// TIA Portal project "sorting and packaging f" (V16)
// Vorlageprojekt für das Buch mit Zielsystem S7-1200

(* hardware
DEVICE "S7-1200-Station_1"  S7-1200 Station
   slot 0: "Baugruppenträger_0"  Rack  V1.0
   slot 1: "PLC_1"  CPU 1211C DC/DC/DC  6ES7 211-1AE40-0XB0  V4.1
*)

// ===== PLC "PLC_1"  CPU 1211C DC/DC/DC =====

VAR_GLOBAL   // PLC tag table "Standard-Variablentabelle"
   "start" AT %I0.0 : Bool;
   "stop" AT %I0.1 : Bool;
   "emergency" AT %I0.2 : Bool;
   "vision1" AT %ID30 : DInt;
   "diff1" AT %I0.4 : Bool;
   "zdownsens1" AT %I0.5 : Bool;
   "box1" AT %I0.7 : Bool;
   "xmovesens1" AT %I1.0 : Bool;
   "rotate1" AT %I1.1 : Bool;
   "diff2" AT %I1.2 : Bool;
   "zdownsens2" AT %I1.3 : Bool;
   "box2" AT %I1.5 : Bool;
   "xmovesens2" AT %I1.6 : Bool;
   "rotate2" AT %I1.7 : Bool;
   "emit1" AT %Q0.0 : Bool;
   "conv1" AT %Q0.1 : Bool;
   "emit2" AT %Q0.2 : Bool;
   "conv2" AT %Q0.3 : Bool;
   "zdown1" AT %Q0.4 : Bool;
   "xmove1" AT %Q0.5 : Bool;
   "turnright1" AT %Q0.6 : Bool;
   "turnleft1" AT %Q0.7 : Bool;
   "zdown2" AT %Q1.0 : Bool;
   "xmove2" AT %Q1.1 : Bool;
   "turnright2" AT %Q1.2 : Bool;
   "turnleft2" AT %Q1.3 : Bool;
   "state" AT %MW500 : Int;
   "Tag_1" AT %M10.4 : Bool;
   "vision1 state" AT %MD38 : DInt;
   "vision2 state" AT %MD42 : DInt;
   "grab1" AT %Q1.4 : Bool;
   "grab2" AT %Q1.5 : Bool;
   "Tag_2" AT %M700.0 : Bool;
   "Tag_3" AT %M700.1 : Bool;
   "vision2" AT %ID34 : DInt;
   "conv" AT %Q2.0 : "udt";
   "diff3" AT %I0.3 : Bool;
   "zdownsens3" AT %I0.6 : Bool;
   "box3" AT %I1.4 : Bool;
   "xmovesens3" AT %I2.0 : Bool;
   "rotate3" AT %I2.1 : Bool;
   "diff4" AT %I2.2 : Bool;
   "zdownsens4" AT %I2.3 : Bool;
   "box4" AT %I2.4 : Bool;
   "xmovesens4" AT %I2.5 : Bool;
   "rotate4" AT %I2.6 : Bool;
   "zdown3" AT %Q2.6 : Bool;
   "xmove3" AT %Q2.7 : Bool;
   "turnright3" AT %Q3.0 : Bool;
   "turnleft3" AT %Q3.1 : Bool;
   "zdown4" AT %Q3.2 : Bool;
   "xmove4" AT %Q3.3 : Bool;
   "turnright4" AT %Q3.4 : Bool;
   "turnleft4" AT %Q3.5 : Bool;
   "grab3" AT %Q3.6 : Bool;
   "grab4" AT %Q3.7 : Bool;
   "Tag_4" AT %M700.2 : Bool;
   "Tag_5" AT %M700.3 : Bool;
   "emitt 3" AT %Q4.0 : Bool;
   "reset" AT %I2.7 : Bool;
   "blue pack conv" AT %Q4.1 : Bool;
   "diff 5" AT %I3.0 : Bool;
   "diff6" AT %I3.1 : Bool;
   "Tag_6" AT %M600.1 : Bool;
   "c1" AT %Q4.2 : Bool;
   "c2" AT %Q4.3 : Bool;
   "c3" AT %Q4.4 : Bool;
   "c4" AT %Q4.5 : Bool;
   "c5" AT %Q4.6 : Bool;
   "c6" AT %Q4.7 : Bool;
   "c7" AT %Q5.0 : Bool;
   "c8" AT %Q5.1 : Bool;
   "c9" AT %Q5.2 : Bool;
   "c10" AT %Q5.3 : Bool;
   "c11" AT %Q5.4 : Bool;
   "c12" AT %Q5.5 : Bool;
   "green x sens" AT %I3.2 : Bool;
   "green z sens" AT %I3.3 : Bool;
   "green rotate" AT %I3.4 : Bool;
   "green box" AT %I3.5 : Bool;
   "green x move" AT %Q5.6 : Bool;
   "green z down" AT %Q5.7 : Bool;
   "green rotate right" AT %Q6.0 : Bool;
   "green rotate left" AT %Q6.1 : Bool;
   "green grab" AT %Q6.2 : Bool;
   "diff7" AT %I3.6 : Bool;
   "diff8" AT %I3.7 : Bool;
   "diff9" AT %I4.0 : Bool;
   "emitter 2 22" AT %Q6.3 : Bool;
   "c13" AT %Q6.4 : Bool;
   "Tag_7" AT %M300.0 : Bool;
   "Tag_8" AT %M300.1 : Bool;
   "palletizer green input" AT %I5.0 : "palletizer input udt";
   "palletize green output" AT %Q7.0 : "palletizer output udt";
   "palletizer blue input" AT %I7.0 : "palletizer input udt";
   "palletizer blue output" AT %Q9.0 : "palletizer output udt";
   "greeen turn table input" AT %I9.0 : "turn table input";
   "blue turn table input" AT %I10.0 : "turn table input";
   "greeen turn table output" AT %Q12.0 : "turn table output";
   "blue turn table output" AT %Q14.0 : "turn table output";
   "warehouse_input" AT %I11.0 : "warehouse input";
   "warehouse_output" AT %Q16.0 : "warehouse output";
   "pos" AT %QD34 : DInt;
END_VAR

TYPE "udt"
   STRUCT
      "conv blue main" : Bool;
      "conv blue second" : Bool;
      "conv green right main" : Bool;
      "conv green right second" : Bool;
      "conv green left main" : Bool;
      "conv green left second" : Bool;
   END_STRUCT;
END_TYPE

TYPE "counters"
   STRUCT
      "counter blue1" : Int := 0;
      "counter reset" : Bool;
      "counter blue 2" : Int := 0;
      "counter total value" : Int := 0;
   END_STRUCT;
END_TYPE

TYPE "flags"
   STRUCT
      "blue forward flag" : Int;
      "blue right flag" : Int;
   END_STRUCT;
END_TYPE

TYPE "palletizer input udt"
   STRUCT
      diff : Bool;
      "pusher sensor" : Bool;
      "load box" : Bool;
      "clamp sensor" : Bool;
      "open plate sensor" : Bool;
      "front limit" : Bool;
      "back limit" : Bool;
      "eleveator moving" : Bool;
      "at entry" : Bool;
      "start palletizer" : Bool;
      "stop palletizer" : Bool;
      "emergency stop palletizer" : Bool;
   END_STRUCT;
END_TYPE

TYPE "palletizer output udt"
   STRUCT
      "box emitter" : Bool;
      "pallet conv out" : Bool;
      c1 : Bool;
      c2 : Bool;
      pusher : Bool;
      "load box" : Bool;
      clamp : Bool;
      "open plate" : Bool;
      "move to limit" : Bool;
      "elevator+" : Bool;
      "elevator-" : Bool;
      "chain+" : Bool;
      "pallet conv" : Bool;
      "paller emiter" : Bool;
   END_STRUCT;
END_TYPE

TYPE "turn table input"
   STRUCT
      "line entry" : Bool;
      "line exit" : Bool;
      "front limit" : Bool;
      "limit 90" : Bool;
      "limit 0" : Bool;
      "line exit finished" : Bool;
   END_STRUCT;
END_TYPE

TYPE "turn table output"
   STRUCT
      ci1 : Bool;
      ci2 : Bool;
      ci3 : Bool;
      "roll+" : Bool;
      "turn table+" : Bool;
      "turn table-" : Bool;
      co1 : Bool;
      "roll-" : Bool;
      "roller stop" : Bool;
   END_STRUCT;
END_TYPE

TYPE "warehouse"
   STRUCT
      id : Array[0..54] of DInt;
      occupied : Array[0..54] of Bool;
   END_STRUCT;
END_TYPE

TYPE "warehouse input"
   STRUCT
      "stop sensor" : Bool;
      "stacker x" : Bool;
      "stacker z" : Bool;
      "stacker right limit" : Bool;
      "stacker left limit" : Bool;
      "stacker middle limit" : Bool;
   END_STRUCT;
END_TYPE

TYPE "warehouse output"
   STRUCT
      cto2 : Bool;
      cto3 : Bool;
      cto4 : Bool;
      cto5 : Bool;
      cto6 : Bool;
      cto7 : Bool;
      cto8 : Bool;
      "loading conv" : Bool;
      right : Bool;
      left : Bool;
      lift : Bool;
      alarm : Bool;
   END_STRUCT;
END_TYPE

DATA_BLOCK "pick and place forward and right_DB"   // DB1
{ S7_Optimized_Access := 'TRUE' }
VERSION : 0.1
// stored: InstanceOfName pick and place forward and right
"pick and place forward and right"
BEGIN
END_DATA_BLOCK

DATA_BLOCK "green package_DB"   // DB2
{ S7_Optimized_Access := 'TRUE' }
VERSION : 0.1
// stored: InstanceOfName green package
"green package"
BEGIN
END_DATA_BLOCK

DATA_BLOCK "packaging right_DB"   // DB4
{ S7_Optimized_Access := 'TRUE' }
VERSION : 0.1
// stored: InstanceOfName packaging right
"packaging right"
BEGIN
END_DATA_BLOCK

DATA_BLOCK "global"   // DB5
{ S7_Optimized_Access := 'TRUE' }
VERSION : 0.1
   VAR
      conv : "udt";
      "palletizer green input" : "palletizer input udt";
      flags : "flags";
      counters : "counters";
      "turn table green input" : "turn table input";
      "turn table green output" : "turn table output";
      warehouse : "warehouse";
   END_VAR
BEGIN
END_DATA_BLOCK

DATA_BLOCK "packaging forward_DB"   // DB6
{ S7_Optimized_Access := 'TRUE' }
VERSION : 0.1
// stored: InstanceOfName packaging forward
"packaging forward"
BEGIN
END_DATA_BLOCK

DATA_BLOCK "pick and place_DB_1"   // DB7
{ S7_Optimized_Access := 'TRUE' }
VERSION : 0.1
// stored: InstanceOfName pick and place forward and left
"pick and place forward and left"
BEGIN
END_DATA_BLOCK

DATA_BLOCK "green palletizer db"   // DB9
{ S7_Optimized_Access := 'TRUE' }
VERSION : 0.1
// stored: InstanceOfName palletizer
"palletizer"
BEGIN
END_DATA_BLOCK

DATA_BLOCK "start conver_DB"   // DB10
{ S7_Optimized_Access := 'TRUE' }
VERSION : 0.1
// stored: InstanceOfName start conver
"start conver"
BEGIN
END_DATA_BLOCK

DATA_BLOCK "blue palletizer db"   // DB11
{ S7_Optimized_Access := 'TRUE' }
VERSION : 0.1
// stored: InstanceOfName palletizer
"palletizer"
BEGIN
END_DATA_BLOCK

DATA_BLOCK "turn table DB"   // DB12
{ S7_Optimized_Access := 'TRUE' }
VERSION : 0.1
// stored: InstanceOfName turn table
"turn table"
BEGIN
END_DATA_BLOCK

DATA_BLOCK "rack_DB"   // DB13
{ S7_Optimized_Access := 'TRUE' }
VERSION : 0.1
// stored: InstanceOfName rack
"rack"
BEGIN
END_DATA_BLOCK

// folder: System blocks/Program resources

DATA_BLOCK "IEC_Counter_0_DB_1"   // DB3
{ S7_Optimized_Access := 'TRUE' }
AUTHOR : Simatic
FAMILY : IEC
NAME : CNTR
VERSION : 1.0
// stored: InstanceOfName IEC_COUNTER
"IEC_COUNTER"
BEGIN
END_DATA_BLOCK

DATA_BLOCK "IEC_Counter_0_DB_2"   // DB8
{ S7_Optimized_Access := 'TRUE' }
AUTHOR : Simatic
FAMILY : IEC
NAME : CNTR
VERSION : 1.0
// stored: InstanceOfName IEC_COUNTER
"IEC_COUNTER"
BEGIN
END_DATA_BLOCK

// folder: (top level)

FUNCTION_BLOCK "pick and place forward and left"   // FB1, LAD
{ S7_Optimized_Access := 'TRUE' }
VERSION : 0.1
   VAR_INPUT
      emergecy : Bool;
      start : Bool;
      stop : Bool;
      vision : DInt;
      diff : Bool;
      "z sensor" : Bool;
      "x sensor" : Bool;
      "box sensor" : Bool;
      rotate : Bool;
   END_VAR
   VAR_OUTPUT
      emiter : Bool;
      conv : Bool;
      "z down" : Bool;
      "x move" : Bool;
      "turn right" : Bool;
      "turn left" : Bool;
      grab : Bool;
   END_VAR
   VAR
      state : Int;
      "last state" : Int;
      "vision state" : DInt;
      "diff state1" : Bool;
      "diff state2" : Bool;
      "box state4" : Bool;
      "box state3" : Bool;
      "box state1" : Bool;
      "box state2" : Bool;
      "zsenor state1" : Bool;
      "xsensor state1" : Bool;
      "xsensor state2" : Bool;
      "xsensor state3" : Bool;
      "xsensor state4" : Bool;
      "xsensor state5" : Bool;
      "zsensor state2" : Bool;
      "zsensor state3" : Bool;
      "zsensor state4" : Bool;
      "zsensor state5" : Bool;
      "zsensor state6" : Bool;
      "rotate state1" : Bool;
      "rotate state2" : Bool;
      "counter reset" : Bool;
      zse1 : Bool;
      zse2 : Bool;
      zse3 : Bool;
      zse4 : Bool;
      zse5 : Bool;
      zse6 : Bool;
      xsens1 : Bool;
      xsens2 : Bool;
      xsens3 : Bool;
      xsens4 : Bool;
      xsens5 : Bool;
      r1 : Bool;
      r2 : Bool;
   END_VAR
   VAR_TEMP   // added for the SCL form of the ladder/FBD networks
      _w1 : Bool;
      _w2 : Bool;
      _w3 : Bool;
      _w4 : Bool;
      _w5 : Bool;
      _w6 : Bool;
      _w7 : Bool;
      _w8 : Bool;
      _w9 : Bool;
      _w10 : Bool;
      _w11 : Bool;
      _w12 : Bool;
      _w13 : Bool;
      _w14 : Bool;
   END_VAR
BEGIN

REGION Network 1
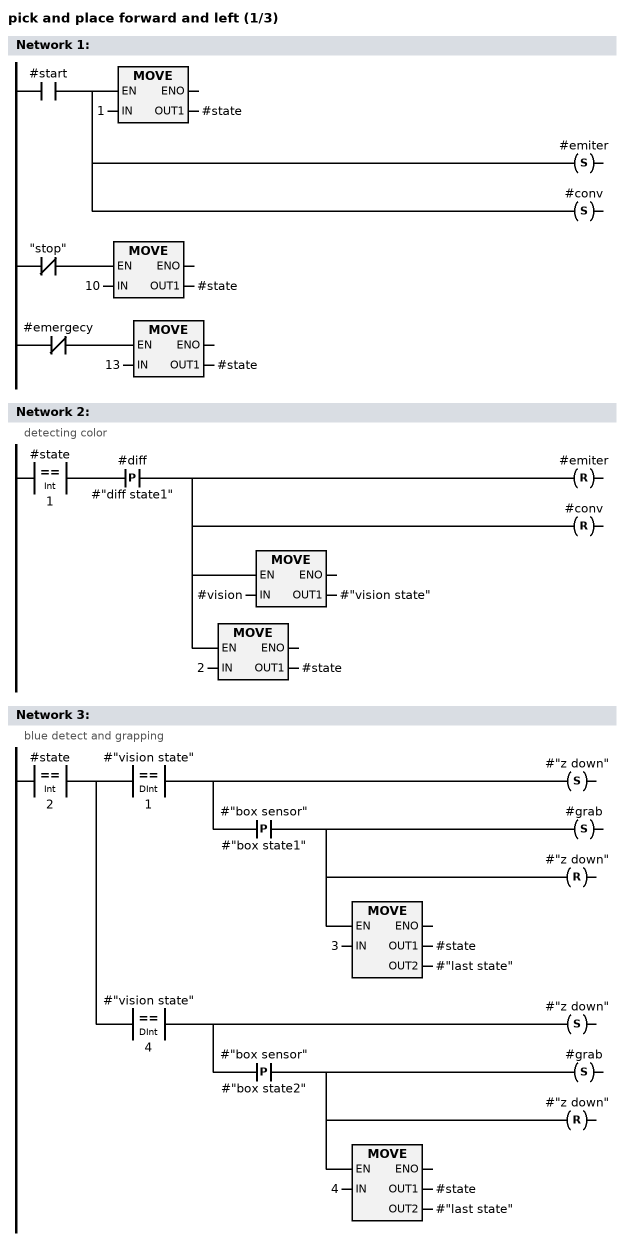
   RUNG wire#powerrail
      Contact( #start )
      wire#w1
      Move(in := 1, out1 => #state)
   END_RUNG
   RUNG wire#w1
      S_Coil( #emiter )
   END_RUNG
   RUNG wire#w1
      S_Coil( #conv )
   END_RUNG
   RUNG wire#powerrail
      I_Contact( "stop" )
      Move(in := 10, out1 => #state)
   END_RUNG
   RUNG wire#powerrail
      I_Contact( #emergecy )
      Move(in := 13, out1 => #state)
   END_RUNG
   // the same network as SCL:
   IF #start THEN
       #state := 1;
       #emiter := TRUE;
       #conv := TRUE;
   END_IF;
   IF NOT "stop" THEN #state := 10; END_IF;
   IF NOT #emergecy THEN #state := 13; END_IF;
END_REGION

REGION Network 2
   // detecting color
   RUNG wire#powerrail
      { S7_Templates := "SrcType := Int" } EQ_Contact(in1 := #state, in2 := 1)
      P_Contact(operand := #diff, bit := #"diff state1")
      wire#w1
      R_Coil( #emiter )
   END_RUNG
   RUNG wire#w1
      R_Coil( #conv )
   END_RUNG
   RUNG wire#w1
      Move(in := #vision, out1 => #"vision state")
   END_RUNG
   RUNG wire#w1
      Move(in := 2, out1 => #state)
   END_RUNG
   // the same network as SCL:
   #_w1 := (#state = 1) AND #diff AND NOT #"diff state1";   // rising edge of #diff
   #"diff state1" := #diff;
   IF #_w1 THEN
       #emiter := FALSE;
       #conv := FALSE;
       #"vision state" := #vision;
       #state := 2;
   END_IF;
END_REGION

REGION Network 3
   // blue detect and grapping
   RUNG wire#powerrail
      { S7_Templates := "SrcType := Int" } EQ_Contact(in1 := #state, in2 := 2)
      wire#w1
      { S7_Templates := "SrcType := DInt" } EQ_Contact(in1 := #"vision state", in2 := 1)
      wire#w2
      S_Coil( #"z down" )
   END_RUNG
   RUNG wire#w2
      P_Contact(operand := #"box sensor", bit := #"box state1")
      wire#w3
      S_Coil( #grab )
   END_RUNG
   RUNG wire#w3
      R_Coil( #"z down" )
   END_RUNG
   RUNG wire#w3
      Move(in := 3, out1 => #state, out2 => #"last state")
   END_RUNG
   RUNG wire#w1
      { S7_Templates := "SrcType := DInt" } EQ_Contact(in1 := #"vision state", in2 := 4)
      wire#w4
      S_Coil( #"z down" )
   END_RUNG
   RUNG wire#w4
      P_Contact(operand := #"box sensor", bit := #"box state2")
      wire#w5
      S_Coil( #grab )
   END_RUNG
   RUNG wire#w5
      R_Coil( #"z down" )
   END_RUNG
   RUNG wire#w5
      Move(in := 4, out1 => #state, out2 => #"last state")
   END_RUNG
   // the same network as SCL:
   #_w1 := #state = 2;
   #_w2 := #_w1 AND (#"vision state" = 1);
   IF #_w2 THEN #"z down" := TRUE; END_IF;
   #_w3 := #_w2 AND #"box sensor" AND NOT #"box state1";   // rising edge of #"box sensor"
   #"box state1" := #"box sensor";
   IF #_w3 THEN
       #grab := TRUE;
       #"z down" := FALSE;
       #state := 3;
       #"last state" := 3;
   END_IF;
   #_w4 := #_w1 AND (#"vision state" = 4);
   IF #_w4 THEN #"z down" := TRUE; END_IF;
   #_w5 := #_w4 AND #"box sensor" AND NOT #"box state2";   // rising edge of #"box sensor"
   #"box state2" := #"box sensor";
   IF #_w5 THEN
       #grab := TRUE;
       #"z down" := FALSE;
       #state := 4;
       #"last state" := 4;
   END_IF;
END_REGION

REGION Network 4
   // blue forward
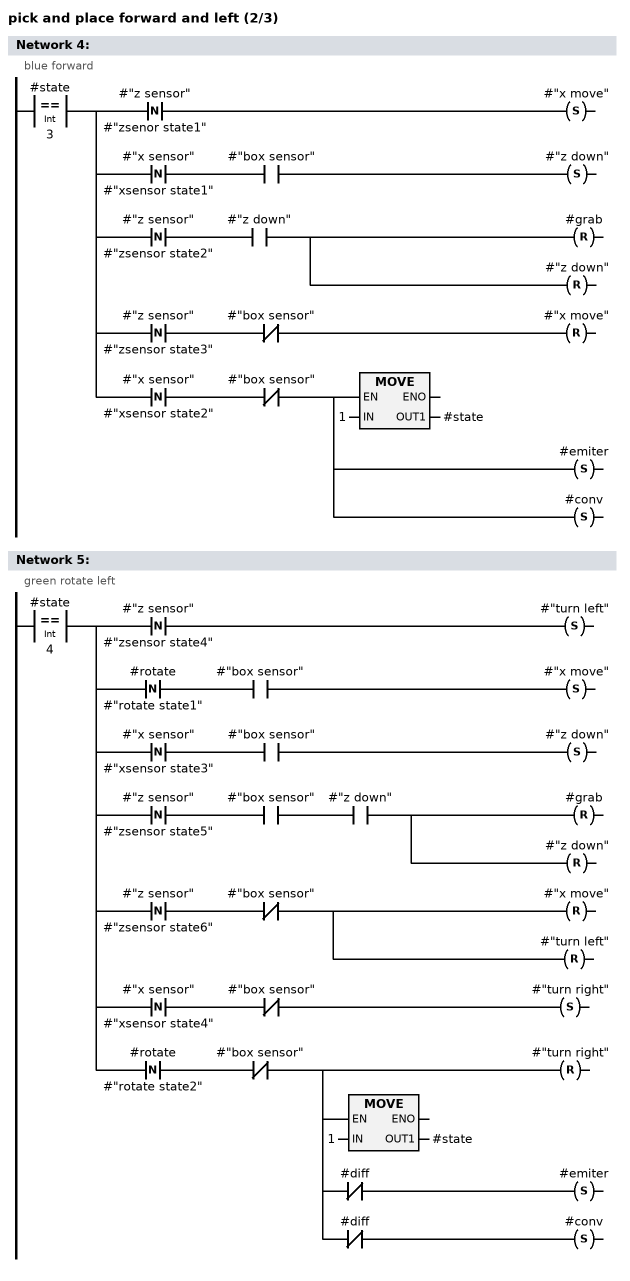
   RUNG wire#powerrail
      { S7_Templates := "SrcType := Int" } EQ_Contact(in1 := #state, in2 := 3)
      wire#w1
      N_Contact(operand := #"z sensor", bit := #"zsenor state1")
      S_Coil( #"x move" )
   END_RUNG
   RUNG wire#w1
      N_Contact(operand := #"x sensor", bit := #"xsensor state1")
      Contact( #"box sensor" )
      S_Coil( #"z down" )
   END_RUNG
   RUNG wire#w1
      N_Contact(operand := #"z sensor", bit := #"zsensor state2")
      Contact( #"z down" )
      wire#w2
      R_Coil( #grab )
   END_RUNG
   RUNG wire#w2
      R_Coil( #"z down" )
   END_RUNG
   RUNG wire#w1
      N_Contact(operand := #"z sensor", bit := #"zsensor state3")
      I_Contact( #"box sensor" )
      R_Coil( #"x move" )
   END_RUNG
   RUNG wire#w1
      N_Contact(operand := #"x sensor", bit := #"xsensor state2")
      I_Contact( #"box sensor" )
      wire#w3
      Move(in := 1, out1 => #state)
   END_RUNG
   RUNG wire#w3
      S_Coil( #emiter )
   END_RUNG
   RUNG wire#w3
      S_Coil( #conv )
   END_RUNG
   // the same network as SCL:
   #_w1 := #state = 3;
   #_w2 := #_w1 AND NOT #"z sensor" AND #"zsenor state1";   // falling edge of #"z sensor"
   #"zsenor state1" := #"z sensor";
   IF #_w2 THEN #"x move" := TRUE; END_IF;
   #_w3 := #_w1 AND NOT #"x sensor" AND #"xsensor state1";   // falling edge of #"x sensor"
   #"xsensor state1" := #"x sensor";
   IF #_w3 AND #"box sensor" THEN #"z down" := TRUE; END_IF;
   #_w4 := #_w1 AND NOT #"z sensor" AND #"zsensor state2";   // falling edge of #"z sensor"
   #"zsensor state2" := #"z sensor";
   IF #_w4 AND #"z down" THEN
       #grab := FALSE;
       #"z down" := FALSE;
   END_IF;
   #_w5 := #_w1 AND NOT #"z sensor" AND #"zsensor state3";   // falling edge of #"z sensor"
   #"zsensor state3" := #"z sensor";
   IF #_w5 AND NOT #"box sensor" THEN #"x move" := FALSE; END_IF;
   #_w6 := #_w1 AND NOT #"x sensor" AND #"xsensor state2";   // falling edge of #"x sensor"
   #"xsensor state2" := #"x sensor";
   IF #_w6 AND NOT #"box sensor" THEN
       #state := 1;
       #emiter := TRUE;
       #conv := TRUE;
   END_IF;
END_REGION

REGION Network 5
   // green rotate left
   RUNG wire#powerrail
      { S7_Templates := "SrcType := Int" } EQ_Contact(in1 := #state, in2 := 4)
      wire#w1
      N_Contact(operand := #"z sensor", bit := #"zsensor state4")
      S_Coil( #"turn left" )
   END_RUNG
   RUNG wire#w1
      N_Contact(operand := #rotate, bit := #"rotate state1")
      Contact( #"box sensor" )
      S_Coil( #"x move" )
   END_RUNG
   RUNG wire#w1
      N_Contact(operand := #"x sensor", bit := #"xsensor state3")
      Contact( #"box sensor" )
      S_Coil( #"z down" )
   END_RUNG
   RUNG wire#w1
      N_Contact(operand := #"z sensor", bit := #"zsensor state5")
      Contact( #"box sensor" )
      Contact( #"z down" )
      wire#w2
      R_Coil( #grab )
   END_RUNG
   RUNG wire#w2
      R_Coil( #"z down" )
   END_RUNG
   RUNG wire#w1
      N_Contact(operand := #"z sensor", bit := #"zsensor state6")
      I_Contact( #"box sensor" )
      wire#w3
      R_Coil( #"x move" )
   END_RUNG
   RUNG wire#w3
      R_Coil( #"turn left" )
   END_RUNG
   RUNG wire#w1
      N_Contact(operand := #"x sensor", bit := #"xsensor state4")
      I_Contact( #"box sensor" )
      S_Coil( #"turn right" )
   END_RUNG
   RUNG wire#w1
      N_Contact(operand := #rotate, bit := #"rotate state2")
      I_Contact( #"box sensor" )
      wire#w4
      R_Coil( #"turn right" )
   END_RUNG
   RUNG wire#w4
      Move(in := 1, out1 => #state)
   END_RUNG
   RUNG wire#w4
      I_Contact( #diff )
      S_Coil( #emiter )
   END_RUNG
   RUNG wire#w4
      I_Contact( #diff )
      S_Coil( #conv )
   END_RUNG
   // the same network as SCL:
   #_w1 := #state = 4;
   #_w2 := #_w1 AND NOT #"z sensor" AND #"zsensor state4";   // falling edge of #"z sensor"
   #"zsensor state4" := #"z sensor";
   IF #_w2 THEN #"turn left" := TRUE; END_IF;
   #_w3 := #_w1 AND NOT #rotate AND #"rotate state1";   // falling edge of #rotate
   #"rotate state1" := #rotate;
   IF #_w3 AND #"box sensor" THEN #"x move" := TRUE; END_IF;
   #_w4 := #_w1 AND NOT #"x sensor" AND #"xsensor state3";   // falling edge of #"x sensor"
   #"xsensor state3" := #"x sensor";
   IF #_w4 AND #"box sensor" THEN #"z down" := TRUE; END_IF;
   #_w5 := #_w1 AND NOT #"z sensor" AND #"zsensor state5";   // falling edge of #"z sensor"
   #"zsensor state5" := #"z sensor";
   IF #_w5 AND #"box sensor" AND #"z down" THEN
       #grab := FALSE;
       #"z down" := FALSE;
   END_IF;
   #_w6 := #_w1 AND NOT #"z sensor" AND #"zsensor state6";   // falling edge of #"z sensor"
   #"zsensor state6" := #"z sensor";
   IF #_w6 AND NOT #"box sensor" THEN
       #"x move" := FALSE;
       #"turn left" := FALSE;
   END_IF;
   #_w7 := #_w1 AND NOT #"x sensor" AND #"xsensor state4";   // falling edge of #"x sensor"
   #"xsensor state4" := #"x sensor";
   IF #_w7 AND NOT #"box sensor" THEN #"turn right" := TRUE; END_IF;
   #_w8 := #_w1 AND NOT #rotate AND #"rotate state2";   // falling edge of #rotate
   #"rotate state2" := #rotate;
   #_w9 := #_w8 AND NOT #"box sensor";
   IF #_w9 THEN
       #"turn right" := FALSE;
       #state := 1;
   END_IF;
   IF #_w9 AND NOT #diff THEN
       #emiter := TRUE;
       #conv := TRUE;
   END_IF;
END_REGION

REGION Network 6
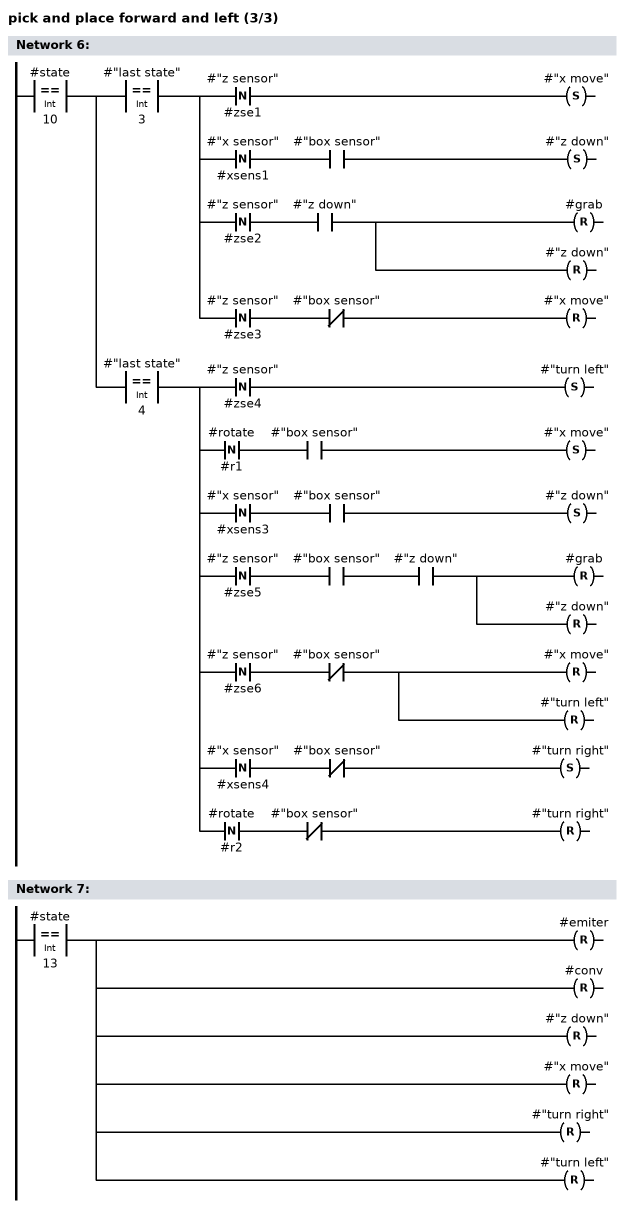
   RUNG wire#powerrail
      { S7_Templates := "SrcType := Int" } EQ_Contact(in1 := #state, in2 := 10)
      wire#w1
      { S7_Templates := "SrcType := Int" } EQ_Contact(in1 := #"last state", in2 := 3)
      wire#w2
      N_Contact(operand := #"z sensor", bit := #zse1)
      S_Coil( #"x move" )
   END_RUNG
   RUNG wire#w2
      N_Contact(operand := #"x sensor", bit := #xsens1)
      Contact( #"box sensor" )
      S_Coil( #"z down" )
   END_RUNG
   RUNG wire#w2
      N_Contact(operand := #"z sensor", bit := #zse2)
      Contact( #"z down" )
      wire#w3
      R_Coil( #grab )
   END_RUNG
   RUNG wire#w3
      R_Coil( #"z down" )
   END_RUNG
   RUNG wire#w2
      N_Contact(operand := #"z sensor", bit := #zse3)
      I_Contact( #"box sensor" )
      R_Coil( #"x move" )
   END_RUNG
   RUNG wire#w1
      { S7_Templates := "SrcType := Int" } EQ_Contact(in1 := #"last state", in2 := 4)
      wire#w4
      N_Contact(operand := #"z sensor", bit := #zse4)
      S_Coil( #"turn left" )
   END_RUNG
   RUNG wire#w4
      N_Contact(operand := #rotate, bit := #r1)
      Contact( #"box sensor" )
      S_Coil( #"x move" )
   END_RUNG
   RUNG wire#w4
      N_Contact(operand := #"x sensor", bit := #xsens3)
      Contact( #"box sensor" )
      S_Coil( #"z down" )
   END_RUNG
   RUNG wire#w4
      N_Contact(operand := #"z sensor", bit := #zse5)
      Contact( #"box sensor" )
      Contact( #"z down" )
      wire#w5
      R_Coil( #grab )
   END_RUNG
   RUNG wire#w5
      R_Coil( #"z down" )
   END_RUNG
   RUNG wire#w4
      N_Contact(operand := #"z sensor", bit := #zse6)
      I_Contact( #"box sensor" )
      wire#w6
      R_Coil( #"x move" )
   END_RUNG
   RUNG wire#w6
      R_Coil( #"turn left" )
   END_RUNG
   RUNG wire#w4
      N_Contact(operand := #"x sensor", bit := #xsens4)
      I_Contact( #"box sensor" )
      S_Coil( #"turn right" )
   END_RUNG
   RUNG wire#w4
      N_Contact(operand := #rotate, bit := #r2)
      I_Contact( #"box sensor" )
      R_Coil( #"turn right" )
   END_RUNG
   // the same network as SCL:
   #_w1 := #state = 10;
   #_w2 := #_w1 AND (#"last state" = 3);
   #_w3 := #_w2 AND NOT #"z sensor" AND #zse1;   // falling edge of #"z sensor"
   #zse1 := #"z sensor";
   IF #_w3 THEN #"x move" := TRUE; END_IF;
   #_w4 := #_w2 AND NOT #"x sensor" AND #xsens1;   // falling edge of #"x sensor"
   #xsens1 := #"x sensor";
   IF #_w4 AND #"box sensor" THEN #"z down" := TRUE; END_IF;
   #_w5 := #_w2 AND NOT #"z sensor" AND #zse2;   // falling edge of #"z sensor"
   #zse2 := #"z sensor";
   IF #_w5 AND #"z down" THEN
       #grab := FALSE;
       #"z down" := FALSE;
   END_IF;
   #_w6 := #_w2 AND NOT #"z sensor" AND #zse3;   // falling edge of #"z sensor"
   #zse3 := #"z sensor";
   IF #_w6 AND NOT #"box sensor" THEN #"x move" := FALSE; END_IF;
   #_w7 := #_w1 AND (#"last state" = 4);
   #_w8 := #_w7 AND NOT #"z sensor" AND #zse4;   // falling edge of #"z sensor"
   #zse4 := #"z sensor";
   IF #_w8 THEN #"turn left" := TRUE; END_IF;
   #_w9 := #_w7 AND NOT #rotate AND #r1;   // falling edge of #rotate
   #r1 := #rotate;
   IF #_w9 AND #"box sensor" THEN #"x move" := TRUE; END_IF;
   #_w10 := #_w7 AND NOT #"x sensor" AND #xsens3;   // falling edge of #"x sensor"
   #xsens3 := #"x sensor";
   IF #_w10 AND #"box sensor" THEN #"z down" := TRUE; END_IF;
   #_w11 := #_w7 AND NOT #"z sensor" AND #zse5;   // falling edge of #"z sensor"
   #zse5 := #"z sensor";
   IF #_w11 AND #"box sensor" AND #"z down" THEN
       #grab := FALSE;
       #"z down" := FALSE;
   END_IF;
   #_w12 := #_w7 AND NOT #"z sensor" AND #zse6;   // falling edge of #"z sensor"
   #zse6 := #"z sensor";
   IF #_w12 AND NOT #"box sensor" THEN
       #"x move" := FALSE;
       #"turn left" := FALSE;
   END_IF;
   #_w13 := #_w7 AND NOT #"x sensor" AND #xsens4;   // falling edge of #"x sensor"
   #xsens4 := #"x sensor";
   IF #_w13 AND NOT #"box sensor" THEN #"turn right" := TRUE; END_IF;
   #_w14 := #_w7 AND NOT #rotate AND #r2;   // falling edge of #rotate
   #r2 := #rotate;
   IF #_w14 AND NOT #"box sensor" THEN #"turn right" := FALSE; END_IF;
END_REGION

REGION Network 7
   RUNG wire#powerrail
      { S7_Templates := "SrcType := Int" } EQ_Contact(in1 := #state, in2 := 13)
      wire#w1
      R_Coil( #emiter )
   END_RUNG
   RUNG wire#w1
      R_Coil( #conv )
   END_RUNG
   RUNG wire#w1
      R_Coil( #"z down" )
   END_RUNG
   RUNG wire#w1
      R_Coil( #"x move" )
   END_RUNG
   RUNG wire#w1
      R_Coil( #"turn right" )
   END_RUNG
   RUNG wire#w1
      R_Coil( #"turn left" )
   END_RUNG
   // the same network as SCL:
   IF #state = 13 THEN
       #emiter := FALSE;
       #conv := FALSE;
       #"z down" := FALSE;
       #"x move" := FALSE;
       #"turn right" := FALSE;
       #"turn left" := FALSE;
   END_IF;
END_REGION
END_FUNCTION_BLOCK

FUNCTION_BLOCK "pick and place forward and right"   // FB2, LAD
{ S7_Optimized_Access := 'TRUE' }
VERSION : 0.1
   VAR_INPUT
      emergecy : Bool;
      start : Bool;
      stop : Bool;
      vision : DInt;
      diff : Bool;
      "z sensor" : Bool;
      "x sensor" : Bool;
      "box sensor" : Bool;
      rotate : Bool;
   END_VAR
   VAR_OUTPUT
      emiter : Bool;
      conv : Bool;
      "z down" : Bool;
      "x move" : Bool;
      "turn right" : Bool;
      "turn left" : Bool;
      grab : Bool;
   END_VAR
   VAR
      state : Int;
      "last state" : Int;
      "vision state" : DInt;
      "diff state1" : Bool;
      "diff state2" : Bool;
      "box state4" : Bool;
      "box state3" : Bool;
      "box state1" : Bool;
      "box state2" : Bool;
      "zsenor state1" : Bool;
      "xsensor state1" : Bool;
      "xsensor state2" : Bool;
      "xsensor state3" : Bool;
      "xsensor state4" : Bool;
      "xsensor state5" : Bool;
      "zsensor state2" : Bool;
      "zsensor state3" : Bool;
      "zsensor state4" : Bool;
      "zsensor state5" : Bool;
      "zsensor state6" : Bool;
      "rotate state1" : Bool;
      "rotate state2" : Bool;
      "counter reset" : Bool;
      final : Bool;
      "timer" : IEC_TIMER;
      "reset timer" : Bool;
      zse1 : Bool;
      zse2 : Bool;
      zse3 : Bool;
      zse4 : Bool;
      zse5 : Bool;
      zse6 : Bool;
      xsens1 : Bool;
      xsens2 : Bool;
      xsens3 : Bool;
      xsens4 : Bool;
      xsens5 : Bool;
      r1 : Bool;
      r2 : Bool;
   END_VAR
   VAR_TEMP   // added for the SCL form of the ladder/FBD networks
      _w1 : Bool;
      _w2 : Bool;
      _w3 : Bool;
      _w4 : Bool;
      _w5 : Bool;
      _w6 : Bool;
      _w7 : Bool;
      _w8 : Bool;
      _w9 : Bool;
      _w10 : Bool;
      _w11 : Bool;
      _w12 : Bool;
      _w13 : Bool;
      _w14 : Bool;
   END_VAR
BEGIN

REGION Network 1
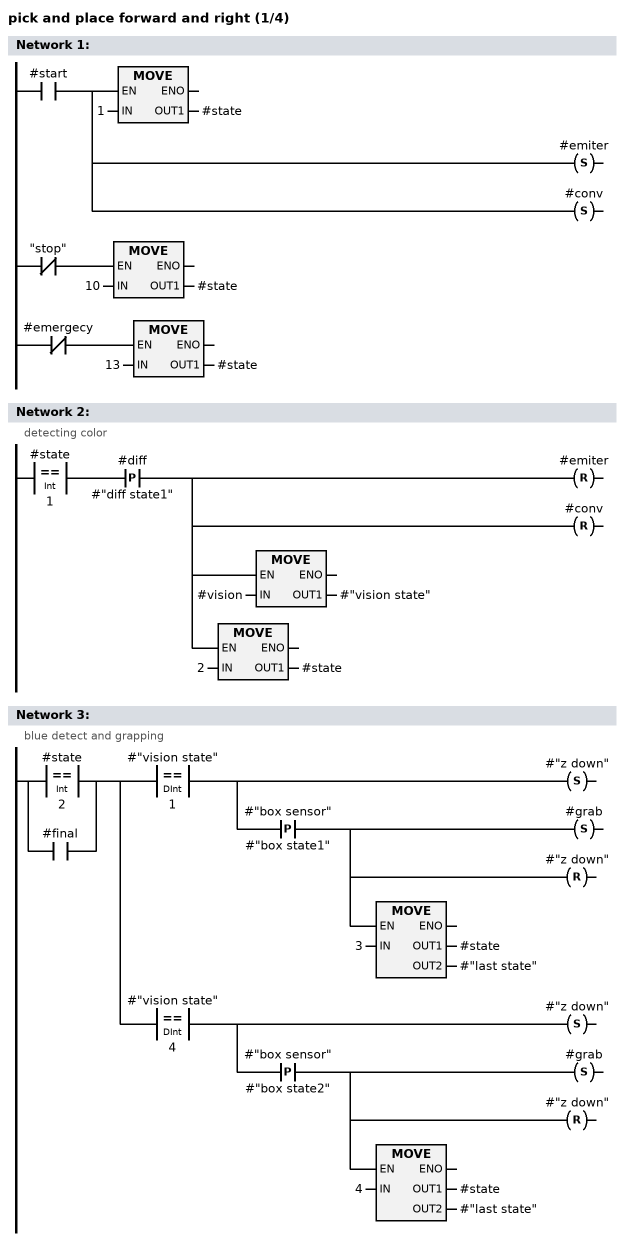
   RUNG wire#powerrail
      Contact( #start )
      wire#w1
      Move(in := 1, out1 => #state)
   END_RUNG
   RUNG wire#w1
      S_Coil( #emiter )
   END_RUNG
   RUNG wire#w1
      S_Coil( #conv )
   END_RUNG
   RUNG wire#powerrail
      I_Contact( "stop" )
      Move(in := 10, out1 => #state)
   END_RUNG
   RUNG wire#powerrail
      I_Contact( #emergecy )
      Move(in := 13, out1 => #state)
   END_RUNG
   // the same network as SCL:
   IF #start THEN
       #state := 1;
       #emiter := TRUE;
       #conv := TRUE;
   END_IF;
   IF NOT "stop" THEN #state := 10; END_IF;
   IF NOT #emergecy THEN #state := 13; END_IF;
END_REGION

REGION Network 2
   // detecting color
   RUNG wire#powerrail
      { S7_Templates := "SrcType := Int" } EQ_Contact(in1 := #state, in2 := 1)
      P_Contact(operand := #diff, bit := #"diff state1")
      wire#w1
      R_Coil( #emiter )
   END_RUNG
   RUNG wire#w1
      R_Coil( #conv )
   END_RUNG
   RUNG wire#w1
      Move(in := #vision, out1 => #"vision state")
   END_RUNG
   RUNG wire#w1
      Move(in := 2, out1 => #state)
   END_RUNG
   // the same network as SCL:
   #_w1 := (#state = 1) AND #diff AND NOT #"diff state1";   // rising edge of #diff
   #"diff state1" := #diff;
   IF #_w1 THEN
       #emiter := FALSE;
       #conv := FALSE;
       #"vision state" := #vision;
       #state := 2;
   END_IF;
END_REGION

REGION Network 3
   // blue detect and grapping
   RUNG wire#powerrail
      { S7_Templates := "SrcType := Int" } EQ_Contact(in1 := #state, in2 := 2)
      wire#w1
      { S7_Templates := "SrcType := DInt" } EQ_Contact(in1 := #"vision state", in2 := 1)
      wire#w2
      S_Coil( #"z down" )
   END_RUNG
   RUNG wire#powerrail
      Contact( #final )
   END_RUNG wire#w1
   RUNG wire#w2
      P_Contact(operand := #"box sensor", bit := #"box state1")
      wire#w3
      S_Coil( #grab )
   END_RUNG
   RUNG wire#w3
      R_Coil( #"z down" )
   END_RUNG
   RUNG wire#w3
      Move(in := 3, out1 => #state, out2 => #"last state")
   END_RUNG
   RUNG wire#w1
      { S7_Templates := "SrcType := DInt" } EQ_Contact(in1 := #"vision state", in2 := 4)
      wire#w4
      S_Coil( #"z down" )
   END_RUNG
   RUNG wire#w4
      P_Contact(operand := #"box sensor", bit := #"box state2")
      wire#w5
      S_Coil( #grab )
   END_RUNG
   RUNG wire#w5
      R_Coil( #"z down" )
   END_RUNG
   RUNG wire#w5
      Move(in := 4, out1 => #state, out2 => #"last state")
   END_RUNG
   // the same network as SCL:
   #_w1 := (#state = 2) OR #final;
   #_w2 := #_w1 AND (#"vision state" = 1);
   IF #_w2 THEN #"z down" := TRUE; END_IF;
   #_w3 := #_w2 AND #"box sensor" AND NOT #"box state1";   // rising edge of #"box sensor"
   #"box state1" := #"box sensor";
   IF #_w3 THEN
       #grab := TRUE;
       #"z down" := FALSE;
       #state := 3;
       #"last state" := 3;
   END_IF;
   #_w4 := #_w1 AND (#"vision state" = 4);
   IF #_w4 THEN #"z down" := TRUE; END_IF;
   #_w5 := #_w4 AND #"box sensor" AND NOT #"box state2";   // rising edge of #"box sensor"
   #"box state2" := #"box sensor";
   IF #_w5 THEN
       #grab := TRUE;
       #"z down" := FALSE;
       #state := 4;
       #"last state" := 4;
   END_IF;
END_REGION

REGION Network 4
   // blue forward
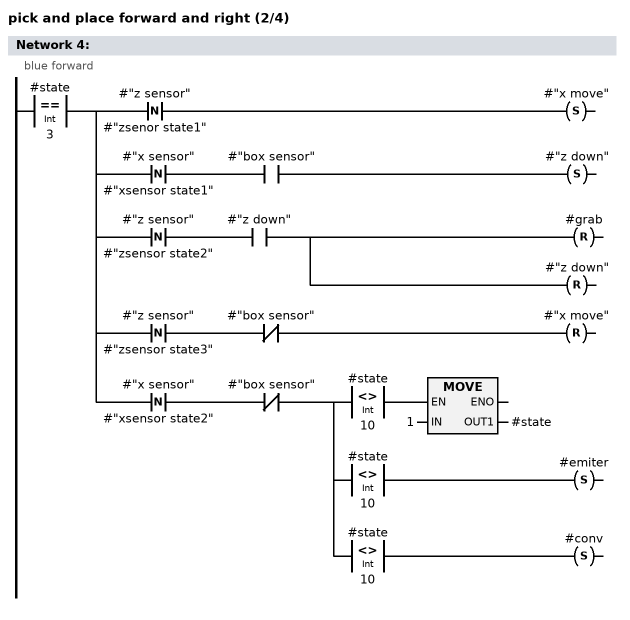
   RUNG wire#powerrail
      { S7_Templates := "SrcType := Int" } EQ_Contact(in1 := #state, in2 := 3)
      wire#w1
      N_Contact(operand := #"z sensor", bit := #"zsenor state1")
      S_Coil( #"x move" )
   END_RUNG
   RUNG wire#w1
      N_Contact(operand := #"x sensor", bit := #"xsensor state1")
      Contact( #"box sensor" )
      S_Coil( #"z down" )
   END_RUNG
   RUNG wire#w1
      N_Contact(operand := #"z sensor", bit := #"zsensor state2")
      Contact( #"z down" )
      wire#w2
      R_Coil( #grab )
   END_RUNG
   RUNG wire#w2
      R_Coil( #"z down" )
   END_RUNG
   RUNG wire#w1
      N_Contact(operand := #"z sensor", bit := #"zsensor state3")
      I_Contact( #"box sensor" )
      R_Coil( #"x move" )
   END_RUNG
   RUNG wire#w1
      N_Contact(operand := #"x sensor", bit := #"xsensor state2")
      I_Contact( #"box sensor" )
      wire#w3
      { S7_Templates := "SrcType := Int" } NE_Contact(in1 := #state, in2 := 10)
      Move(in := 1, out1 => #state)
   END_RUNG
   RUNG wire#w3
      { S7_Templates := "SrcType := Int" } NE_Contact(in1 := #state, in2 := 10)
      S_Coil( #emiter )
   END_RUNG
   RUNG wire#w3
      { S7_Templates := "SrcType := Int" } NE_Contact(in1 := #state, in2 := 10)
      S_Coil( #conv )
   END_RUNG
   // the same network as SCL:
   #_w1 := #state = 3;
   #_w2 := #_w1 AND NOT #"z sensor" AND #"zsenor state1";   // falling edge of #"z sensor"
   #"zsenor state1" := #"z sensor";
   IF #_w2 THEN #"x move" := TRUE; END_IF;
   #_w3 := #_w1 AND NOT #"x sensor" AND #"xsensor state1";   // falling edge of #"x sensor"
   #"xsensor state1" := #"x sensor";
   IF #_w3 AND #"box sensor" THEN #"z down" := TRUE; END_IF;
   #_w4 := #_w1 AND NOT #"z sensor" AND #"zsensor state2";   // falling edge of #"z sensor"
   #"zsensor state2" := #"z sensor";
   IF #_w4 AND #"z down" THEN
       #grab := FALSE;
       #"z down" := FALSE;
   END_IF;
   #_w5 := #_w1 AND NOT #"z sensor" AND #"zsensor state3";   // falling edge of #"z sensor"
   #"zsensor state3" := #"z sensor";
   IF #_w5 AND NOT #"box sensor" THEN #"x move" := FALSE; END_IF;
   #_w6 := #_w1 AND NOT #"x sensor" AND #"xsensor state2";   // falling edge of #"x sensor"
   #"xsensor state2" := #"x sensor";
   #_w7 := #_w6 AND NOT #"box sensor";
   IF #_w7 AND (#state <> 10) THEN #state := 1; END_IF;
   IF #_w7 AND (#state <> 10) THEN
       #emiter := TRUE;
       #conv := TRUE;
   END_IF;
END_REGION

REGION Network 5
   // green rotate left
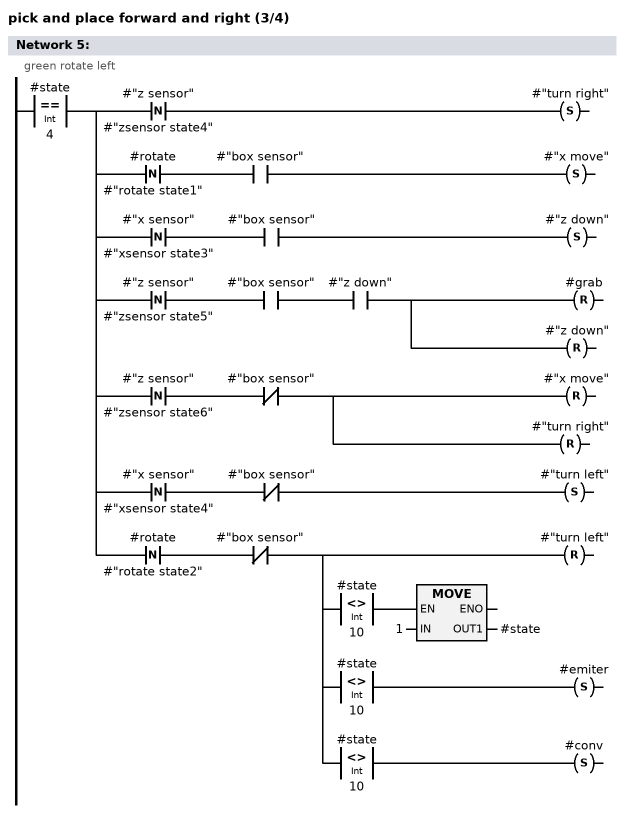
   RUNG wire#powerrail
      { S7_Templates := "SrcType := Int" } EQ_Contact(in1 := #state, in2 := 4)
      wire#w1
      N_Contact(operand := #"z sensor", bit := #"zsensor state4")
      S_Coil( #"turn right" )
   END_RUNG
   RUNG wire#w1
      N_Contact(operand := #rotate, bit := #"rotate state1")
      Contact( #"box sensor" )
      S_Coil( #"x move" )
   END_RUNG
   RUNG wire#w1
      N_Contact(operand := #"x sensor", bit := #"xsensor state3")
      Contact( #"box sensor" )
      S_Coil( #"z down" )
   END_RUNG
   RUNG wire#w1
      N_Contact(operand := #"z sensor", bit := #"zsensor state5")
      Contact( #"box sensor" )
      Contact( #"z down" )
      wire#w2
      R_Coil( #grab )
   END_RUNG
   RUNG wire#w2
      R_Coil( #"z down" )
   END_RUNG
   RUNG wire#w1
      N_Contact(operand := #"z sensor", bit := #"zsensor state6")
      I_Contact( #"box sensor" )
      wire#w3
      R_Coil( #"x move" )
   END_RUNG
   RUNG wire#w3
      R_Coil( #"turn right" )
   END_RUNG
   RUNG wire#w1
      N_Contact(operand := #"x sensor", bit := #"xsensor state4")
      I_Contact( #"box sensor" )
      S_Coil( #"turn left" )
   END_RUNG
   RUNG wire#w1
      N_Contact(operand := #rotate, bit := #"rotate state2")
      I_Contact( #"box sensor" )
      wire#w4
      R_Coil( #"turn left" )
   END_RUNG
   RUNG wire#w4
      { S7_Templates := "SrcType := Int" } NE_Contact(in1 := #state, in2 := 10)
      Move(in := 1, out1 => #state)
   END_RUNG
   RUNG wire#w4
      { S7_Templates := "SrcType := Int" } NE_Contact(in1 := #state, in2 := 10)
      S_Coil( #emiter )
   END_RUNG
   RUNG wire#w4
      { S7_Templates := "SrcType := Int" } NE_Contact(in1 := #state, in2 := 10)
      S_Coil( #conv )
   END_RUNG
   // the same network as SCL:
   #_w1 := #state = 4;
   #_w2 := #_w1 AND NOT #"z sensor" AND #"zsensor state4";   // falling edge of #"z sensor"
   #"zsensor state4" := #"z sensor";
   IF #_w2 THEN #"turn right" := TRUE; END_IF;
   #_w3 := #_w1 AND NOT #rotate AND #"rotate state1";   // falling edge of #rotate
   #"rotate state1" := #rotate;
   IF #_w3 AND #"box sensor" THEN #"x move" := TRUE; END_IF;
   #_w4 := #_w1 AND NOT #"x sensor" AND #"xsensor state3";   // falling edge of #"x sensor"
   #"xsensor state3" := #"x sensor";
   IF #_w4 AND #"box sensor" THEN #"z down" := TRUE; END_IF;
   #_w5 := #_w1 AND NOT #"z sensor" AND #"zsensor state5";   // falling edge of #"z sensor"
   #"zsensor state5" := #"z sensor";
   IF #_w5 AND #"box sensor" AND #"z down" THEN
       #grab := FALSE;
       #"z down" := FALSE;
   END_IF;
   #_w6 := #_w1 AND NOT #"z sensor" AND #"zsensor state6";   // falling edge of #"z sensor"
   #"zsensor state6" := #"z sensor";
   IF #_w6 AND NOT #"box sensor" THEN
       #"x move" := FALSE;
       #"turn right" := FALSE;
   END_IF;
   #_w7 := #_w1 AND NOT #"x sensor" AND #"xsensor state4";   // falling edge of #"x sensor"
   #"xsensor state4" := #"x sensor";
   IF #_w7 AND NOT #"box sensor" THEN #"turn left" := TRUE; END_IF;
   #_w8 := #_w1 AND NOT #rotate AND #"rotate state2";   // falling edge of #rotate
   #"rotate state2" := #rotate;
   #_w9 := #_w8 AND NOT #"box sensor";
   IF #_w9 THEN #"turn left" := FALSE; END_IF;
   IF #_w9 AND (#state <> 10) THEN #state := 1; END_IF;
   IF #_w9 AND (#state <> 10) THEN
       #emiter := TRUE;
       #conv := TRUE;
   END_IF;
END_REGION

REGION Network 6
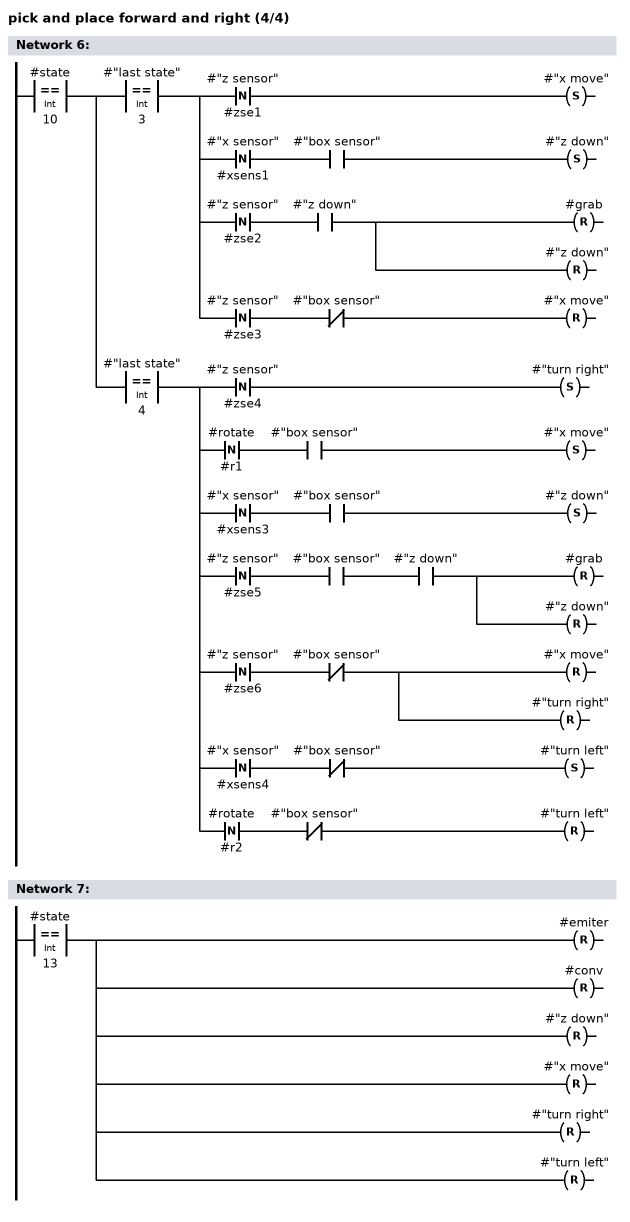
   RUNG wire#powerrail
      { S7_Templates := "SrcType := Int" } EQ_Contact(in1 := #state, in2 := 10)
      wire#w1
      { S7_Templates := "SrcType := Int" } EQ_Contact(in1 := #"last state", in2 := 3)
      wire#w2
      N_Contact(operand := #"z sensor", bit := #zse1)
      S_Coil( #"x move" )
   END_RUNG
   RUNG wire#w2
      N_Contact(operand := #"x sensor", bit := #xsens1)
      Contact( #"box sensor" )
      S_Coil( #"z down" )
   END_RUNG
   RUNG wire#w2
      N_Contact(operand := #"z sensor", bit := #zse2)
      Contact( #"z down" )
      wire#w3
      R_Coil( #grab )
   END_RUNG
   RUNG wire#w3
      R_Coil( #"z down" )
   END_RUNG
   RUNG wire#w2
      N_Contact(operand := #"z sensor", bit := #zse3)
      I_Contact( #"box sensor" )
      R_Coil( #"x move" )
   END_RUNG
   RUNG wire#w1
      { S7_Templates := "SrcType := Int" } EQ_Contact(in1 := #"last state", in2 := 4)
      wire#w4
      N_Contact(operand := #"z sensor", bit := #zse4)
      S_Coil( #"turn right" )
   END_RUNG
   RUNG wire#w4
      N_Contact(operand := #rotate, bit := #r1)
      Contact( #"box sensor" )
      S_Coil( #"x move" )
   END_RUNG
   RUNG wire#w4
      N_Contact(operand := #"x sensor", bit := #xsens3)
      Contact( #"box sensor" )
      S_Coil( #"z down" )
   END_RUNG
   RUNG wire#w4
      N_Contact(operand := #"z sensor", bit := #zse5)
      Contact( #"box sensor" )
      Contact( #"z down" )
      wire#w5
      R_Coil( #grab )
   END_RUNG
   RUNG wire#w5
      R_Coil( #"z down" )
   END_RUNG
   RUNG wire#w4
      N_Contact(operand := #"z sensor", bit := #zse6)
      I_Contact( #"box sensor" )
      wire#w6
      R_Coil( #"x move" )
   END_RUNG
   RUNG wire#w6
      R_Coil( #"turn right" )
   END_RUNG
   RUNG wire#w4
      N_Contact(operand := #"x sensor", bit := #xsens4)
      I_Contact( #"box sensor" )
      S_Coil( #"turn left" )
   END_RUNG
   RUNG wire#w4
      N_Contact(operand := #rotate, bit := #r2)
      I_Contact( #"box sensor" )
      R_Coil( #"turn left" )
   END_RUNG
   // the same network as SCL:
   #_w1 := #state = 10;
   #_w2 := #_w1 AND (#"last state" = 3);
   #_w3 := #_w2 AND NOT #"z sensor" AND #zse1;   // falling edge of #"z sensor"
   #zse1 := #"z sensor";
   IF #_w3 THEN #"x move" := TRUE; END_IF;
   #_w4 := #_w2 AND NOT #"x sensor" AND #xsens1;   // falling edge of #"x sensor"
   #xsens1 := #"x sensor";
   IF #_w4 AND #"box sensor" THEN #"z down" := TRUE; END_IF;
   #_w5 := #_w2 AND NOT #"z sensor" AND #zse2;   // falling edge of #"z sensor"
   #zse2 := #"z sensor";
   IF #_w5 AND #"z down" THEN
       #grab := FALSE;
       #"z down" := FALSE;
   END_IF;
   #_w6 := #_w2 AND NOT #"z sensor" AND #zse3;   // falling edge of #"z sensor"
   #zse3 := #"z sensor";
   IF #_w6 AND NOT #"box sensor" THEN #"x move" := FALSE; END_IF;
   #_w7 := #_w1 AND (#"last state" = 4);
   #_w8 := #_w7 AND NOT #"z sensor" AND #zse4;   // falling edge of #"z sensor"
   #zse4 := #"z sensor";
   IF #_w8 THEN #"turn right" := TRUE; END_IF;
   #_w9 := #_w7 AND NOT #rotate AND #r1;   // falling edge of #rotate
   #r1 := #rotate;
   IF #_w9 AND #"box sensor" THEN #"x move" := TRUE; END_IF;
   #_w10 := #_w7 AND NOT #"x sensor" AND #xsens3;   // falling edge of #"x sensor"
   #xsens3 := #"x sensor";
   IF #_w10 AND #"box sensor" THEN #"z down" := TRUE; END_IF;
   #_w11 := #_w7 AND NOT #"z sensor" AND #zse5;   // falling edge of #"z sensor"
   #zse5 := #"z sensor";
   IF #_w11 AND #"box sensor" AND #"z down" THEN
       #grab := FALSE;
       #"z down" := FALSE;
   END_IF;
   #_w12 := #_w7 AND NOT #"z sensor" AND #zse6;   // falling edge of #"z sensor"
   #zse6 := #"z sensor";
   IF #_w12 AND NOT #"box sensor" THEN
       #"x move" := FALSE;
       #"turn right" := FALSE;
   END_IF;
   #_w13 := #_w7 AND NOT #"x sensor" AND #xsens4;   // falling edge of #"x sensor"
   #xsens4 := #"x sensor";
   IF #_w13 AND NOT #"box sensor" THEN #"turn left" := TRUE; END_IF;
   #_w14 := #_w7 AND NOT #rotate AND #r2;   // falling edge of #rotate
   #r2 := #rotate;
   IF #_w14 AND NOT #"box sensor" THEN #"turn left" := FALSE; END_IF;
END_REGION

REGION Network 7
   RUNG wire#powerrail
      { S7_Templates := "SrcType := Int" } EQ_Contact(in1 := #state, in2 := 13)
      wire#w1
      R_Coil( #emiter )
   END_RUNG
   RUNG wire#w1
      R_Coil( #conv )
   END_RUNG
   RUNG wire#w1
      R_Coil( #"z down" )
   END_RUNG
   RUNG wire#w1
      R_Coil( #"x move" )
   END_RUNG
   RUNG wire#w1
      R_Coil( #"turn right" )
   END_RUNG
   RUNG wire#w1
      R_Coil( #"turn left" )
   END_RUNG
   // the same network as SCL:
   IF #state = 13 THEN
       #emiter := FALSE;
       #conv := FALSE;
       #"z down" := FALSE;
       #"x move" := FALSE;
       #"turn right" := FALSE;
       #"turn left" := FALSE;
   END_IF;
END_REGION
END_FUNCTION_BLOCK

FUNCTION_BLOCK "packaging right"   // FB3, LAD
{ S7_Optimized_Access := 'TRUE' }
VERSION : 0.1
   VAR_INPUT
      emergecy : Bool;
      start : Bool;
      stop : Bool;
      diff : Bool;
      "z sensor" : Bool;
      "x sensor" : Bool;
      "box sensor" : Bool;
      rotate : Bool;
      "counter reset" : Bool;
   END_VAR
   VAR_OUTPUT
      conv1 : Bool;
      conv2 : Bool;
      "z down" : Bool;
      "x move" : Bool;
      "turn right" : Bool;
      "turn left" : Bool;
      grab : Bool;
   END_VAR
   VAR
      state : Int;
      "last state" : Int;
      "vision state" : Bool;
      "diff state1" : Bool;
      "diff state2" : Bool;
      "box state4" : Bool;
      "box state3" : Bool;
      "box state1" : Bool;
      "box state2" : Bool;
      "zsenor state1" : Bool;
      "xsensor state1" : Bool;
      "xsensor state2" : Bool;
      "xsensor state3" : Bool;
      "xsensor state4" : Bool;
      "xsensor state5" : Bool;
      "zsensor state2" : Bool;
      "zsensor state3" : Bool;
      "zsensor state4" : Bool;
      "zsensor state5" : Bool;
      "zsensor state6" : Bool;
      "rotate state1" : Bool;
      "rotate state2" : Bool;
      zse1 : Bool;
      zse2 : Bool;
      zse3 : Bool;
      zse4 : Bool;
      zse5 : Bool;
      zse6 : Bool;
      xsens1 : Bool;
      xsens2 : Bool;
      xsens3 : Bool;
      xsens4 : Bool;
      xsens5 : Bool;
      r1 : Bool;
      r2 : Bool;
      flags : "flags";
   END_VAR
   VAR_TEMP   // added for the SCL form of the ladder/FBD networks
      _w1 : Bool;
      _w2 : Bool;
      _w3 : Bool;
      _w4 : Bool;
      _w5 : Bool;
      _w6 : Bool;
      _w7 : Bool;
      _w8 : Bool;
      _w9 : Bool;
      _w10 : Bool;
   END_VAR
BEGIN

REGION Network 2
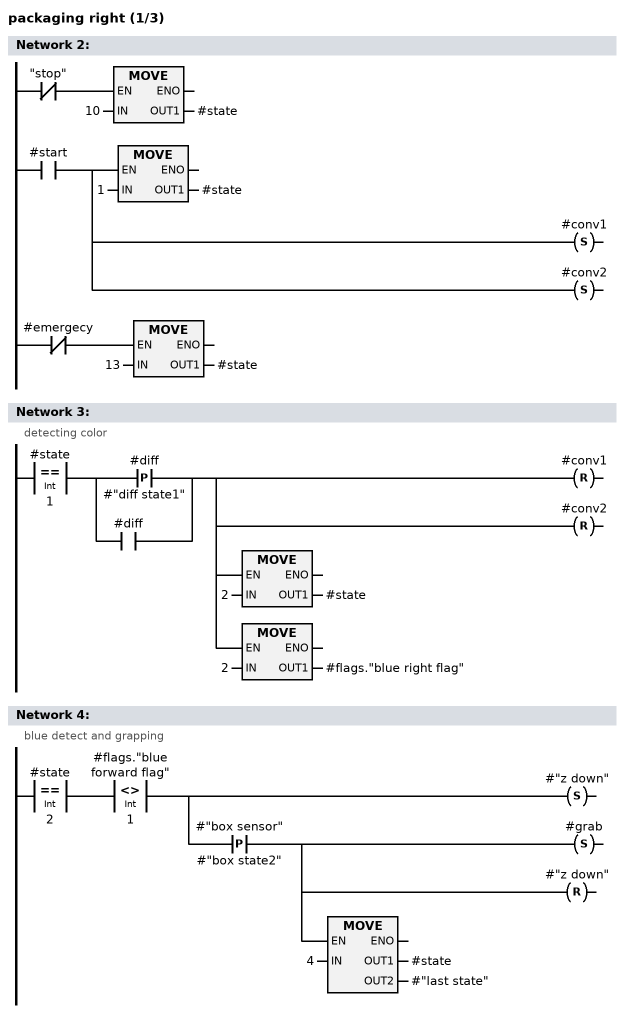
   RUNG wire#powerrail
      I_Contact( "stop" )
      Move(in := 10, out1 => #state)
   END_RUNG
   RUNG wire#powerrail
      Contact( #start )
      wire#w1
      Move(in := 1, out1 => #state)
   END_RUNG
   RUNG wire#w1
      S_Coil( #conv1 )
   END_RUNG
   RUNG wire#w1
      S_Coil( #conv2 )
   END_RUNG
   RUNG wire#powerrail
      I_Contact( #emergecy )
      Move(in := 13, out1 => #state)
   END_RUNG
   // the same network as SCL:
   IF NOT "stop" THEN #state := 10; END_IF;
   IF #start THEN
       #state := 1;
       #conv1 := TRUE;
       #conv2 := TRUE;
   END_IF;
   IF NOT #emergecy THEN #state := 13; END_IF;
END_REGION

REGION Network 3
   // detecting color
   RUNG wire#powerrail
      { S7_Templates := "SrcType := Int" } EQ_Contact(in1 := #state, in2 := 1)
      wire#w1
      P_Contact(operand := #diff, bit := #"diff state1")
      wire#w2
      R_Coil( #conv1 )
   END_RUNG
   RUNG wire#w1
      Contact( #diff )
   END_RUNG wire#w2
   RUNG wire#w2
      R_Coil( #conv2 )
   END_RUNG
   RUNG wire#w2
      Move(in := 2, out1 => #state)
   END_RUNG
   RUNG wire#w2
      Move(in := 2, out1 => #flags."blue right flag")
   END_RUNG
   // the same network as SCL:
   #_w1 := (#state = 1) AND #diff AND NOT #"diff state1";   // rising edge of #diff
   #"diff state1" := #diff;
   IF #_w1 OR ((#state = 1) AND #diff) THEN
       #conv1 := FALSE;
       #conv2 := FALSE;
   END_IF;
   #_w2 := #_w1 OR ((#state = 1) AND #diff);
   IF #_w2 THEN
       #state := 2;
       #flags."blue right flag" := 2;
   END_IF;
END_REGION

REGION Network 4
   // blue detect and grapping
   RUNG wire#powerrail
      { S7_Templates := "SrcType := Int" } EQ_Contact(in1 := #state, in2 := 2)
      { S7_Templates := "SrcType := Int" } NE_Contact(in1 := #flags."blue forward flag", in2 := 1)
      wire#w1
      S_Coil( #"z down" )
   END_RUNG
   RUNG wire#w1
      P_Contact(operand := #"box sensor", bit := #"box state2")
      wire#w2
      S_Coil( #grab )
   END_RUNG
   RUNG wire#w2
      R_Coil( #"z down" )
   END_RUNG
   RUNG wire#w2
      Move(in := 4, out1 => #state, out2 => #"last state")
   END_RUNG
   // the same network as SCL:
   #_w1 := (#state = 2) AND (#flags."blue forward flag" <> 1);
   IF #_w1 THEN #"z down" := TRUE; END_IF;
   #_w2 := #_w1 AND #"box sensor" AND NOT #"box state2";   // rising edge of #"box sensor"
   #"box state2" := #"box sensor";
   IF #_w2 THEN
       #grab := TRUE;
       #"z down" := FALSE;
       #state := 4;
       #"last state" := 4;
   END_IF;
END_REGION

REGION Network 5
   // green rotate left
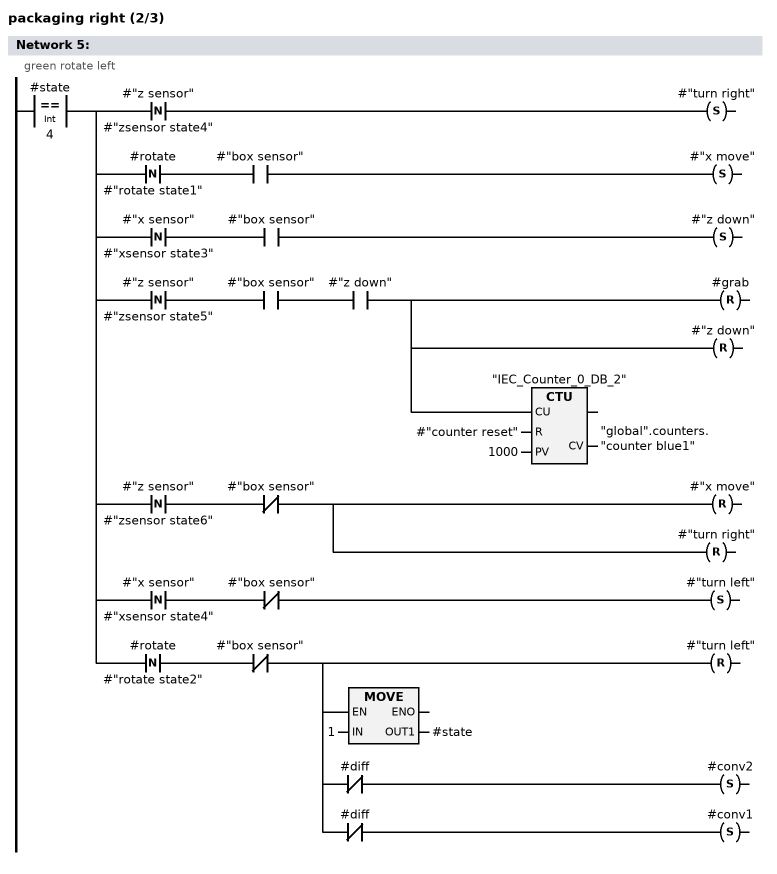
   #_w1 := #state = 4;
   #_w2 := #_w1 AND NOT #"z sensor" AND #"zsensor state4";   // falling edge of #"z sensor"
   #"zsensor state4" := #"z sensor";
   IF #_w2 THEN #"turn right" := TRUE; END_IF;
   #_w3 := #_w1 AND NOT #rotate AND #"rotate state1";   // falling edge of #rotate
   #"rotate state1" := #rotate;
   IF #_w3 AND #"box sensor" THEN #"x move" := TRUE; END_IF;
   #_w4 := #_w1 AND NOT #"x sensor" AND #"xsensor state3";   // falling edge of #"x sensor"
   #"xsensor state3" := #"x sensor";
   IF #_w4 AND #"box sensor" THEN #"z down" := TRUE; END_IF;
   #_w5 := #_w1 AND NOT #"z sensor" AND #"zsensor state5";   // falling edge of #"z sensor"
   #"zsensor state5" := #"z sensor";
   #_w6 := #_w5 AND #"box sensor" AND #"z down";
   IF #_w6 THEN
       #grab := FALSE;
       #"z down" := FALSE;
   END_IF;
   "IEC_Counter_0_DB_2".CTU(CU := #_w6,
                           R := #"counter reset",
                           PV := 1000,
                           CV => "global".counters."counter blue1");
   #_w7 := #_w1 AND NOT #"z sensor" AND #"zsensor state6";   // falling edge of #"z sensor"
   #"zsensor state6" := #"z sensor";
   IF #_w7 AND NOT #"box sensor" THEN
       #"x move" := FALSE;
       #"turn right" := FALSE;
   END_IF;
   #_w8 := #_w1 AND NOT #"x sensor" AND #"xsensor state4";   // falling edge of #"x sensor"
   #"xsensor state4" := #"x sensor";
   IF #_w8 AND NOT #"box sensor" THEN #"turn left" := TRUE; END_IF;
   #_w9 := #_w1 AND NOT #rotate AND #"rotate state2";   // falling edge of #rotate
   #"rotate state2" := #rotate;
   #_w10 := #_w9 AND NOT #"box sensor";
   IF #_w10 THEN
       #"turn left" := FALSE;
       #state := 1;
   END_IF;
   IF #_w10 AND NOT #diff THEN
       #conv2 := TRUE;
       #conv1 := TRUE;
   END_IF;
END_REGION

REGION Network 6
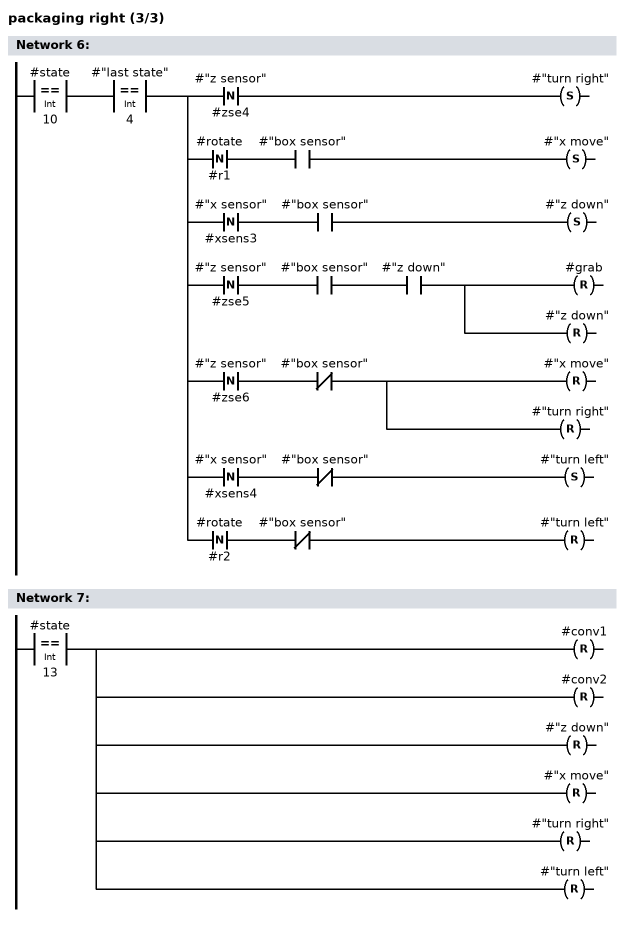
   RUNG wire#powerrail
      { S7_Templates := "SrcType := Int" } EQ_Contact(in1 := #state, in2 := 10)
      { S7_Templates := "SrcType := Int" } EQ_Contact(in1 := #"last state", in2 := 4)
      wire#w1
      N_Contact(operand := #"z sensor", bit := #zse4)
      S_Coil( #"turn right" )
   END_RUNG
   RUNG wire#w1
      N_Contact(operand := #rotate, bit := #r1)
      Contact( #"box sensor" )
      S_Coil( #"x move" )
   END_RUNG
   RUNG wire#w1
      N_Contact(operand := #"x sensor", bit := #xsens3)
      Contact( #"box sensor" )
      S_Coil( #"z down" )
   END_RUNG
   RUNG wire#w1
      N_Contact(operand := #"z sensor", bit := #zse5)
      Contact( #"box sensor" )
      Contact( #"z down" )
      wire#w2
      R_Coil( #grab )
   END_RUNG
   RUNG wire#w2
      R_Coil( #"z down" )
   END_RUNG
   RUNG wire#w1
      N_Contact(operand := #"z sensor", bit := #zse6)
      I_Contact( #"box sensor" )
      wire#w3
      R_Coil( #"x move" )
   END_RUNG
   RUNG wire#w3
      R_Coil( #"turn right" )
   END_RUNG
   RUNG wire#w1
      N_Contact(operand := #"x sensor", bit := #xsens4)
      I_Contact( #"box sensor" )
      S_Coil( #"turn left" )
   END_RUNG
   RUNG wire#w1
      N_Contact(operand := #rotate, bit := #r2)
      I_Contact( #"box sensor" )
      R_Coil( #"turn left" )
   END_RUNG
   // the same network as SCL:
   #_w1 := (#state = 10) AND (#"last state" = 4);
   #_w2 := #_w1 AND NOT #"z sensor" AND #zse4;   // falling edge of #"z sensor"
   #zse4 := #"z sensor";
   IF #_w2 THEN #"turn right" := TRUE; END_IF;
   #_w3 := #_w1 AND NOT #rotate AND #r1;   // falling edge of #rotate
   #r1 := #rotate;
   IF #_w3 AND #"box sensor" THEN #"x move" := TRUE; END_IF;
   #_w4 := #_w1 AND NOT #"x sensor" AND #xsens3;   // falling edge of #"x sensor"
   #xsens3 := #"x sensor";
   IF #_w4 AND #"box sensor" THEN #"z down" := TRUE; END_IF;
   #_w5 := #_w1 AND NOT #"z sensor" AND #zse5;   // falling edge of #"z sensor"
   #zse5 := #"z sensor";
   IF #_w5 AND #"box sensor" AND #"z down" THEN
       #grab := FALSE;
       #"z down" := FALSE;
   END_IF;
   #_w6 := #_w1 AND NOT #"z sensor" AND #zse6;   // falling edge of #"z sensor"
   #zse6 := #"z sensor";
   IF #_w6 AND NOT #"box sensor" THEN
       #"x move" := FALSE;
       #"turn right" := FALSE;
   END_IF;
   #_w7 := #_w1 AND NOT #"x sensor" AND #xsens4;   // falling edge of #"x sensor"
   #xsens4 := #"x sensor";
   IF #_w7 AND NOT #"box sensor" THEN #"turn left" := TRUE; END_IF;
   #_w8 := #_w1 AND NOT #rotate AND #r2;   // falling edge of #rotate
   #r2 := #rotate;
   IF #_w8 AND NOT #"box sensor" THEN #"turn left" := FALSE; END_IF;
END_REGION

REGION Network 7
   RUNG wire#powerrail
      { S7_Templates := "SrcType := Int" } EQ_Contact(in1 := #state, in2 := 13)
      wire#w1
      R_Coil( #conv1 )
   END_RUNG
   RUNG wire#w1
      R_Coil( #conv2 )
   END_RUNG
   RUNG wire#w1
      R_Coil( #"z down" )
   END_RUNG
   RUNG wire#w1
      R_Coil( #"x move" )
   END_RUNG
   RUNG wire#w1
      R_Coil( #"turn right" )
   END_RUNG
   RUNG wire#w1
      R_Coil( #"turn left" )
   END_RUNG
   // the same network as SCL:
   IF #state = 13 THEN
       #conv1 := FALSE;
       #conv2 := FALSE;
       #"z down" := FALSE;
       #"x move" := FALSE;
       #"turn right" := FALSE;
       #"turn left" := FALSE;
   END_IF;
END_REGION
END_FUNCTION_BLOCK

FUNCTION_BLOCK "packaging forward"   // FB4, LAD
{ S7_Optimized_Access := 'TRUE' }
VERSION : 0.1
   VAR_INPUT
      emergecy : Bool;
      start : Bool;
      stop : Bool;
      diff : Bool;
      "z sensor" : Bool;
      "x sensor" : Bool;
      "box sensor" : Bool;
      rotate : Bool;
      "counter reset" : Bool;
   END_VAR
   VAR_OUTPUT
      conv1 : Bool;
      conv2 : Bool;
      "z down" : Bool;
      "x move" : Bool;
      "turn right" : Bool;
      "turn left" : Bool;
      grab : Bool;
   END_VAR
   VAR
      state : Int;
      "last state" : Int;
      "vision state" : Bool;
      "diff state1" : Bool;
      "diff state2" : Bool;
      "box state4" : Bool;
      "box state3" : Bool;
      "box state1" : Bool;
      "box state2" : Bool;
      "zsenor state1" : Bool;
      "xsensor state1" : Bool;
      "xsensor state2" : Bool;
      "xsensor state3" : Bool;
      "xsensor state4" : Bool;
      "xsensor state5" : Bool;
      "zsensor state2" : Bool;
      "zsensor state3" : Bool;
      "zsensor state4" : Bool;
      "zsensor state5" : Bool;
      "zsensor state6" : Bool;
      "rotate state1" : Bool;
      "rotate state2" : Bool;
      zse1 : Bool;
      zse2 : Bool;
      zse3 : Bool;
      zse4 : Bool;
      zse5 : Bool;
      zse6 : Bool;
      xsens1 : Bool;
      xsens2 : Bool;
      xsens3 : Bool;
      xsens4 : Bool;
      xsens5 : Bool;
      r1 : Bool;
      r2 : Bool;
      flags : "flags";
   END_VAR
   VAR_TEMP   // added for the SCL form of the ladder/FBD networks
      _w1 : Bool;
      _w2 : Bool;
      _w3 : Bool;
      _w4 : Bool;
      _w5 : Bool;
      _w6 : Bool;
      _w7 : Bool;
      _w8 : Bool;
   END_VAR
BEGIN

REGION Network 2
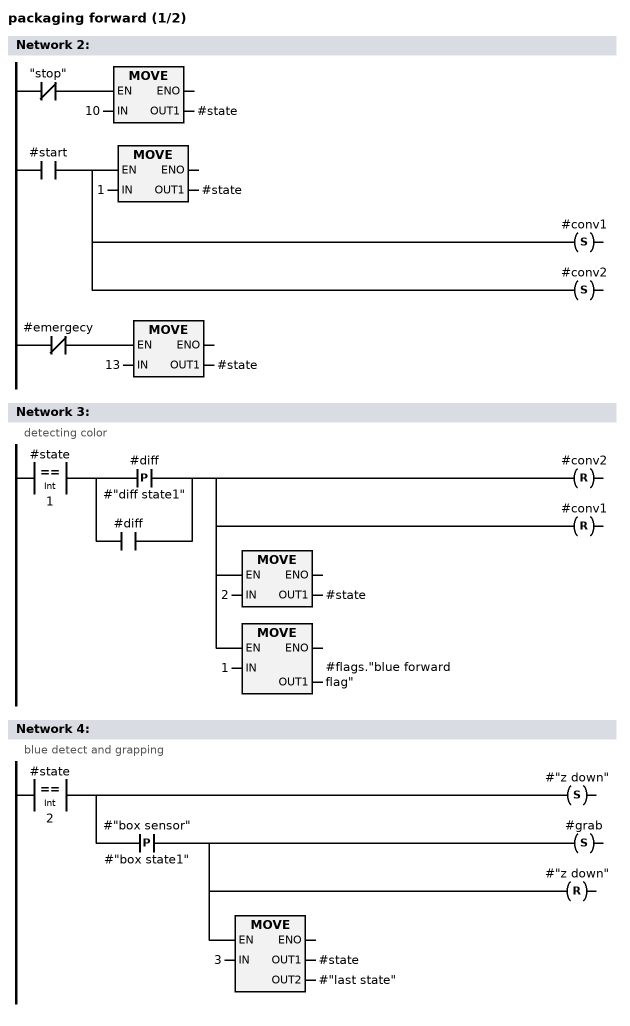
   RUNG wire#powerrail
      I_Contact( "stop" )
      Move(in := 10, out1 => #state)
   END_RUNG
   RUNG wire#powerrail
      Contact( #start )
      wire#w1
      Move(in := 1, out1 => #state)
   END_RUNG
   RUNG wire#w1
      S_Coil( #conv1 )
   END_RUNG
   RUNG wire#w1
      S_Coil( #conv2 )
   END_RUNG
   RUNG wire#powerrail
      I_Contact( #emergecy )
      Move(in := 13, out1 => #state)
   END_RUNG
   // the same network as SCL:
   IF NOT "stop" THEN #state := 10; END_IF;
   IF #start THEN
       #state := 1;
       #conv1 := TRUE;
       #conv2 := TRUE;
   END_IF;
   IF NOT #emergecy THEN #state := 13; END_IF;
END_REGION

REGION Network 3
   // detecting color
   RUNG wire#powerrail
      { S7_Templates := "SrcType := Int" } EQ_Contact(in1 := #state, in2 := 1)
      wire#w1
      P_Contact(operand := #diff, bit := #"diff state1")
      wire#w2
      R_Coil( #conv2 )
   END_RUNG
   RUNG wire#w1
      Contact( #diff )
   END_RUNG wire#w2
   RUNG wire#w2
      R_Coil( #conv1 )
   END_RUNG
   RUNG wire#w2
      Move(in := 2, out1 => #state)
   END_RUNG
   RUNG wire#w2
      Move(in := 1, out1 => #flags."blue forward flag")
   END_RUNG
   // the same network as SCL:
   #_w1 := (#state = 1) AND #diff AND NOT #"diff state1";   // rising edge of #diff
   #"diff state1" := #diff;
   IF #_w1 OR ((#state = 1) AND #diff) THEN
       #conv2 := FALSE;
       #conv1 := FALSE;
   END_IF;
   #_w2 := #_w1 OR ((#state = 1) AND #diff);
   IF #_w2 THEN
       #state := 2;
       #flags."blue forward flag" := 1;
   END_IF;
END_REGION

REGION Network 4
   // blue detect and grapping
   RUNG wire#powerrail
      { S7_Templates := "SrcType := Int" } EQ_Contact(in1 := #state, in2 := 2)
      wire#w1
      S_Coil( #"z down" )
   END_RUNG
   RUNG wire#w1
      P_Contact(operand := #"box sensor", bit := #"box state1")
      wire#w2
      S_Coil( #grab )
   END_RUNG
   RUNG wire#w2
      R_Coil( #"z down" )
   END_RUNG
   RUNG wire#w2
      Move(in := 3, out1 => #state, out2 => #"last state")
   END_RUNG
   // the same network as SCL:
   #_w1 := #state = 2;
   IF #_w1 THEN #"z down" := TRUE; END_IF;
   #_w2 := #_w1 AND #"box sensor" AND NOT #"box state1";   // rising edge of #"box sensor"
   #"box state1" := #"box sensor";
   IF #_w2 THEN
       #grab := TRUE;
       #"z down" := FALSE;
       #state := 3;
       #"last state" := 3;
   END_IF;
END_REGION

REGION Network 5
   // blue forward
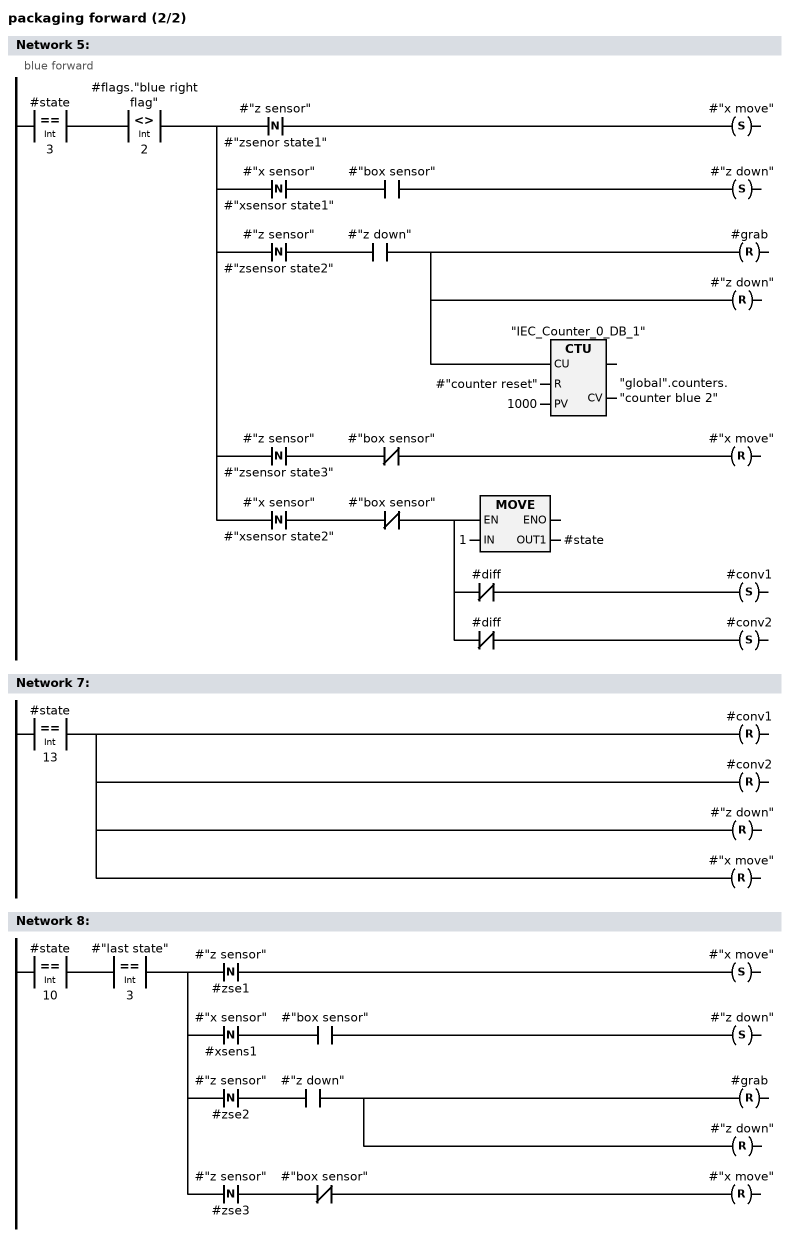
   #_w1 := (#state = 3) AND (#flags."blue right flag" <> 2);
   #_w2 := #_w1 AND NOT #"z sensor" AND #"zsenor state1";   // falling edge of #"z sensor"
   #"zsenor state1" := #"z sensor";
   IF #_w2 THEN #"x move" := TRUE; END_IF;
   #_w3 := #_w1 AND NOT #"x sensor" AND #"xsensor state1";   // falling edge of #"x sensor"
   #"xsensor state1" := #"x sensor";
   IF #_w3 AND #"box sensor" THEN #"z down" := TRUE; END_IF;
   #_w4 := #_w1 AND NOT #"z sensor" AND #"zsensor state2";   // falling edge of #"z sensor"
   #"zsensor state2" := #"z sensor";
   #_w5 := #_w4 AND #"z down";
   IF #_w5 THEN
       #grab := FALSE;
       #"z down" := FALSE;
   END_IF;
   "IEC_Counter_0_DB_1".CTU(CU := #_w5,
                           R := #"counter reset",
                           PV := 1000,
                           CV => "global".counters."counter blue 2");
   #_w6 := #_w1 AND NOT #"z sensor" AND #"zsensor state3";   // falling edge of #"z sensor"
   #"zsensor state3" := #"z sensor";
   IF #_w6 AND NOT #"box sensor" THEN #"x move" := FALSE; END_IF;
   #_w7 := #_w1 AND NOT #"x sensor" AND #"xsensor state2";   // falling edge of #"x sensor"
   #"xsensor state2" := #"x sensor";
   #_w8 := #_w7 AND NOT #"box sensor";
   IF #_w8 THEN #state := 1; END_IF;
   IF #_w8 AND NOT #diff THEN
       #conv1 := TRUE;
       #conv2 := TRUE;
   END_IF;
END_REGION

REGION Network 7
   RUNG wire#powerrail
      { S7_Templates := "SrcType := Int" } EQ_Contact(in1 := #state, in2 := 13)
      wire#w1
      R_Coil( #conv1 )
   END_RUNG
   RUNG wire#w1
      R_Coil( #conv2 )
   END_RUNG
   RUNG wire#w1
      R_Coil( #"z down" )
   END_RUNG
   RUNG wire#w1
      R_Coil( #"x move" )
   END_RUNG
   // the same network as SCL:
   IF #state = 13 THEN
       #conv1 := FALSE;
       #conv2 := FALSE;
       #"z down" := FALSE;
       #"x move" := FALSE;
   END_IF;
END_REGION

REGION Network 8
   RUNG wire#powerrail
      { S7_Templates := "SrcType := Int" } EQ_Contact(in1 := #state, in2 := 10)
      { S7_Templates := "SrcType := Int" } EQ_Contact(in1 := #"last state", in2 := 3)
      wire#w1
      N_Contact(operand := #"z sensor", bit := #zse1)
      S_Coil( #"x move" )
   END_RUNG
   RUNG wire#w1
      N_Contact(operand := #"x sensor", bit := #xsens1)
      Contact( #"box sensor" )
      S_Coil( #"z down" )
   END_RUNG
   RUNG wire#w1
      N_Contact(operand := #"z sensor", bit := #zse2)
      Contact( #"z down" )
      wire#w2
      R_Coil( #grab )
   END_RUNG
   RUNG wire#w2
      R_Coil( #"z down" )
   END_RUNG
   RUNG wire#w1
      N_Contact(operand := #"z sensor", bit := #zse3)
      I_Contact( #"box sensor" )
      R_Coil( #"x move" )
   END_RUNG
   // the same network as SCL:
   #_w1 := (#state = 10) AND (#"last state" = 3);
   #_w2 := #_w1 AND NOT #"z sensor" AND #zse1;   // falling edge of #"z sensor"
   #zse1 := #"z sensor";
   IF #_w2 THEN #"x move" := TRUE; END_IF;
   #_w3 := #_w1 AND NOT #"x sensor" AND #xsens1;   // falling edge of #"x sensor"
   #xsens1 := #"x sensor";
   IF #_w3 AND #"box sensor" THEN #"z down" := TRUE; END_IF;
   #_w4 := #_w1 AND NOT #"z sensor" AND #zse2;   // falling edge of #"z sensor"
   #zse2 := #"z sensor";
   IF #_w4 AND #"z down" THEN
       #grab := FALSE;
       #"z down" := FALSE;
   END_IF;
   #_w5 := #_w1 AND NOT #"z sensor" AND #zse3;   // falling edge of #"z sensor"
   #zse3 := #"z sensor";
   IF #_w5 AND NOT #"box sensor" THEN #"x move" := FALSE; END_IF;
END_REGION
END_FUNCTION_BLOCK

FUNCTION_BLOCK "green package"   // FB5, LAD
{ S7_Optimized_Access := 'TRUE' }
VERSION : 0.1
   VAR_INPUT
      emergecy : Bool;
      start : Bool;
      stop : Bool;
      diff1 : Bool;
      diff2 : Bool;
      diff3 : Bool;
      "z sensor" : Bool;
      "x sensor" : Bool;
      "box sensor" : Bool;
      rotate : Bool;
      "global counter reset" : Bool;
   END_VAR
   VAR_OUTPUT
      conv1 : Bool;
      conv2 : Bool;
      "z down" : Bool;
      "x move" : Bool;
      "turn right" : Bool;
      "turn left" : Bool;
      grab : Bool;
      emiter : Bool;
   END_VAR
   VAR
      state : Int;
      "last state" : Int;
      "vision state" : Bool;
      "diff state1" : Bool;
      "diff state2" : Bool;
      "box state4" : Bool;
      "box state3" : Bool;
      "box state1" : Bool;
      "box state2" : Bool;
      "zsenor state1" : Bool;
      "xsensor state1" : Bool;
      "xsensor state2" : Bool;
      "xsensor state3" : Bool;
      "xsensor state4" : Bool;
      "xsensor state5" : Bool;
      "zsensor state2" : Bool;
      "zsensor state3" : Bool;
      "zsensor state4" : Bool;
      "zsensor state5" : Bool;
      "zsensor state6" : Bool;
      "rotate state1" : Bool;
      "rotate state2" : Bool;
      "diff3 state" : Bool;
      "counter reset" : Bool;
      counter1 : IEC_UCOUNTER;
      zse1 : Bool;
      zse2 : Bool;
      zse3 : Bool;
      zse4 : Bool;
      zse5 : Bool;
      zse6 : Bool;
      xsens1 : Bool;
      xsens2 : Bool;
      xsens3 : Bool;
      xsens4 : Bool;
      xsens5 : Bool;
      r1 : Bool;
      r2 : Bool;
   END_VAR
   VAR_TEMP   // added for the SCL form of the ladder/FBD networks
      _w1 : Bool;
      _w2 : Bool;
      _w3 : Bool;
      _w4 : Bool;
      _w5 : Bool;
      _w6 : Bool;
      _w7 : Bool;
      _w8 : Bool;
      _w9 : Bool;
      _w10 : Bool;
   END_VAR
BEGIN

REGION Network 1
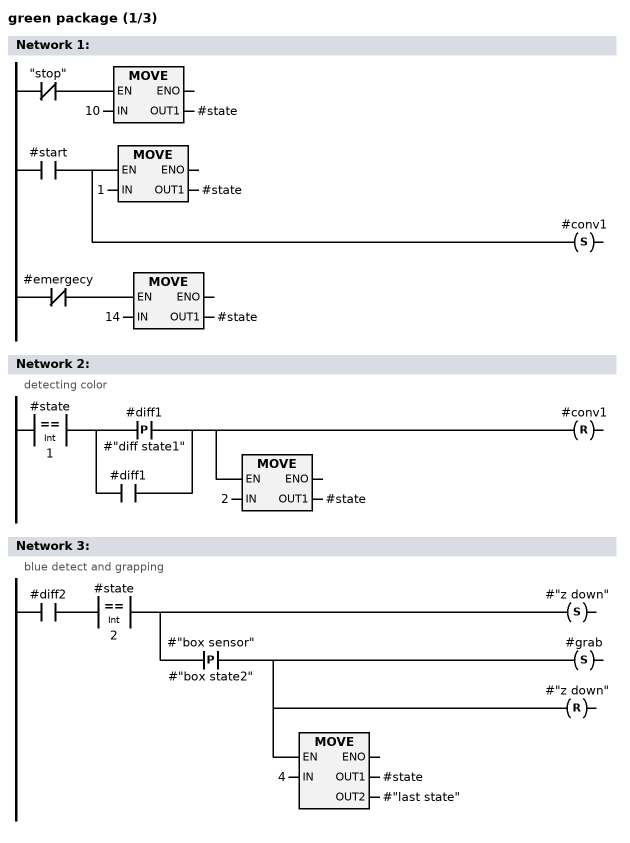
   RUNG wire#powerrail
      I_Contact( "stop" )
      Move(in := 10, out1 => #state)
   END_RUNG
   RUNG wire#powerrail
      Contact( #start )
      wire#w1
      Move(in := 1, out1 => #state)
   END_RUNG
   RUNG wire#w1
      S_Coil( #conv1 )
   END_RUNG
   RUNG wire#powerrail
      I_Contact( #emergecy )
      Move(in := 14, out1 => #state)
   END_RUNG
   // the same network as SCL:
   IF NOT "stop" THEN #state := 10; END_IF;
   IF #start THEN
       #state := 1;
       #conv1 := TRUE;
   END_IF;
   IF NOT #emergecy THEN #state := 14; END_IF;
END_REGION

REGION Network 2
   // detecting color
   RUNG wire#powerrail
      { S7_Templates := "SrcType := Int" } EQ_Contact(in1 := #state, in2 := 1)
      wire#w1
      P_Contact(operand := #diff1, bit := #"diff state1")
      wire#w2
      R_Coil( #conv1 )
   END_RUNG
   RUNG wire#w1
      Contact( #diff1 )
   END_RUNG wire#w2
   RUNG wire#w2
      Move(in := 2, out1 => #state)
   END_RUNG
   // the same network as SCL:
   #_w1 := (#state = 1) AND #diff1 AND NOT #"diff state1";   // rising edge of #diff1
   #"diff state1" := #diff1;
   IF #_w1 OR ((#state = 1) AND #diff1) THEN
       #conv1 := FALSE;
       #state := 2;
   END_IF;
END_REGION

REGION Network 3
   // blue detect and grapping
   RUNG wire#powerrail
      Contact( #diff2 )
      { S7_Templates := "SrcType := Int" } EQ_Contact(in1 := #state, in2 := 2)
      wire#w1
      S_Coil( #"z down" )
   END_RUNG
   RUNG wire#w1
      P_Contact(operand := #"box sensor", bit := #"box state2")
      wire#w2
      S_Coil( #grab )
   END_RUNG
   RUNG wire#w2
      R_Coil( #"z down" )
   END_RUNG
   RUNG wire#w2
      Move(in := 4, out1 => #state, out2 => #"last state")
   END_RUNG
   // the same network as SCL:
   #_w1 := #diff2 AND (#state = 2);
   IF #_w1 THEN #"z down" := TRUE; END_IF;
   #_w2 := #_w1 AND #"box sensor" AND NOT #"box state2";   // rising edge of #"box sensor"
   #"box state2" := #"box sensor";
   IF #_w2 THEN
       #grab := TRUE;
       #"z down" := FALSE;
       #state := 4;
       #"last state" := 4;
   END_IF;
END_REGION

REGION Network 4
   // green rotate left
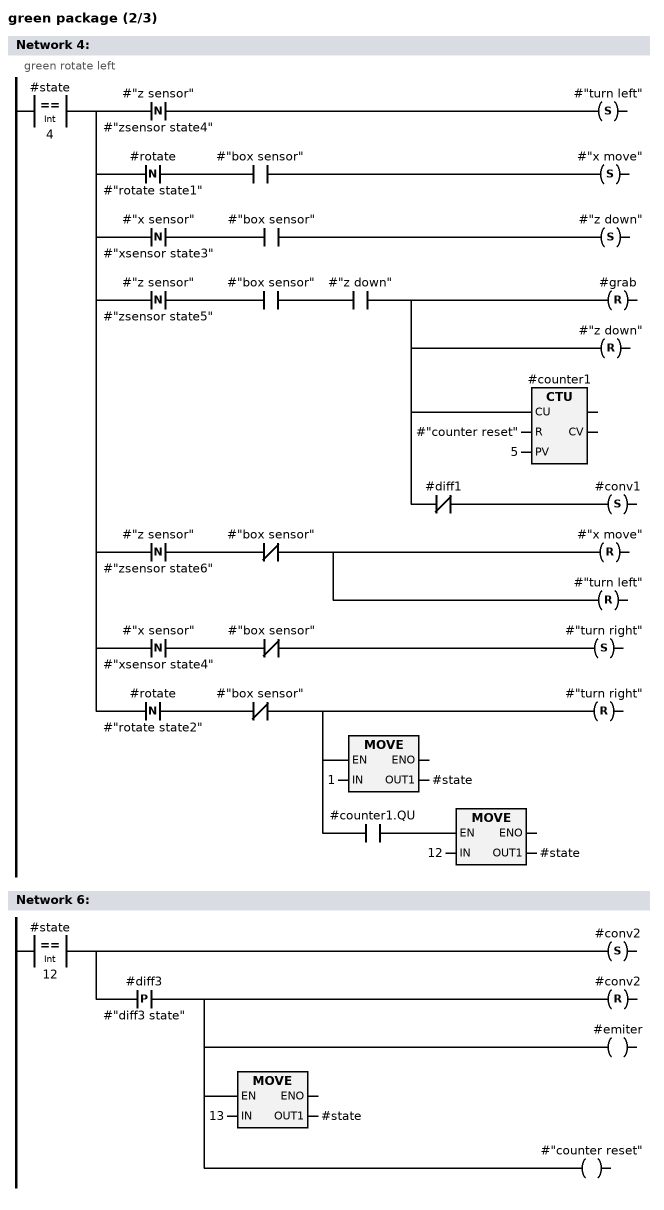
   #_w1 := #state = 4;
   #_w2 := #_w1 AND NOT #"z sensor" AND #"zsensor state4";   // falling edge of #"z sensor"
   #"zsensor state4" := #"z sensor";
   IF #_w2 THEN #"turn left" := TRUE; END_IF;
   #_w3 := #_w1 AND NOT #rotate AND #"rotate state1";   // falling edge of #rotate
   #"rotate state1" := #rotate;
   IF #_w3 AND #"box sensor" THEN #"x move" := TRUE; END_IF;
   #_w4 := #_w1 AND NOT #"x sensor" AND #"xsensor state3";   // falling edge of #"x sensor"
   #"xsensor state3" := #"x sensor";
   IF #_w4 AND #"box sensor" THEN #"z down" := TRUE; END_IF;
   #_w5 := #_w1 AND NOT #"z sensor" AND #"zsensor state5";   // falling edge of #"z sensor"
   #"zsensor state5" := #"z sensor";
   #_w6 := #_w5 AND #"box sensor" AND #"z down";
   IF #_w6 THEN
       #grab := FALSE;
       #"z down" := FALSE;
   END_IF;
   #counter1.CTU(CU := #_w6, R := #"counter reset", PV := 5);
   IF #_w6 AND NOT #diff1 THEN #conv1 := TRUE; END_IF;
   #_w7 := #_w1 AND NOT #"z sensor" AND #"zsensor state6";   // falling edge of #"z sensor"
   #"zsensor state6" := #"z sensor";
   IF #_w7 AND NOT #"box sensor" THEN
       #"x move" := FALSE;
       #"turn left" := FALSE;
   END_IF;
   #_w8 := #_w1 AND NOT #"x sensor" AND #"xsensor state4";   // falling edge of #"x sensor"
   #"xsensor state4" := #"x sensor";
   IF #_w8 AND NOT #"box sensor" THEN #"turn right" := TRUE; END_IF;
   #_w9 := #_w1 AND NOT #rotate AND #"rotate state2";   // falling edge of #rotate
   #"rotate state2" := #rotate;
   #_w10 := #_w9 AND NOT #"box sensor";
   IF #_w10 THEN
       #"turn right" := FALSE;
       #state := 1;
   END_IF;
   IF #_w10 AND #counter1.QU THEN #state := 12; END_IF;
END_REGION

REGION Network 6
   RUNG wire#powerrail
      { S7_Templates := "SrcType := Int" } EQ_Contact(in1 := #state, in2 := 12)
      wire#w1
      S_Coil( #conv2 )
   END_RUNG
   RUNG wire#w1
      P_Contact(operand := #diff3, bit := #"diff3 state")
      wire#w2
      R_Coil( #conv2 )
   END_RUNG
   RUNG wire#w2
      Coil( #emiter )
   END_RUNG
   RUNG wire#w2
      Move(in := 13, out1 => #state)
   END_RUNG
   RUNG wire#w2
      Coil( #"counter reset" )
   END_RUNG
   // the same network as SCL:
   #_w1 := #state = 12;
   IF #_w1 THEN #conv2 := TRUE; END_IF;
   #_w2 := #_w1 AND #diff3 AND NOT #"diff3 state";   // rising edge of #diff3
   #"diff3 state" := #diff3;
   IF #_w2 THEN #conv2 := FALSE; END_IF;
   #emiter := #_w2;
   IF #_w2 THEN #state := 13; END_IF;
   #"counter reset" := #_w2;
END_REGION

REGION Network 7
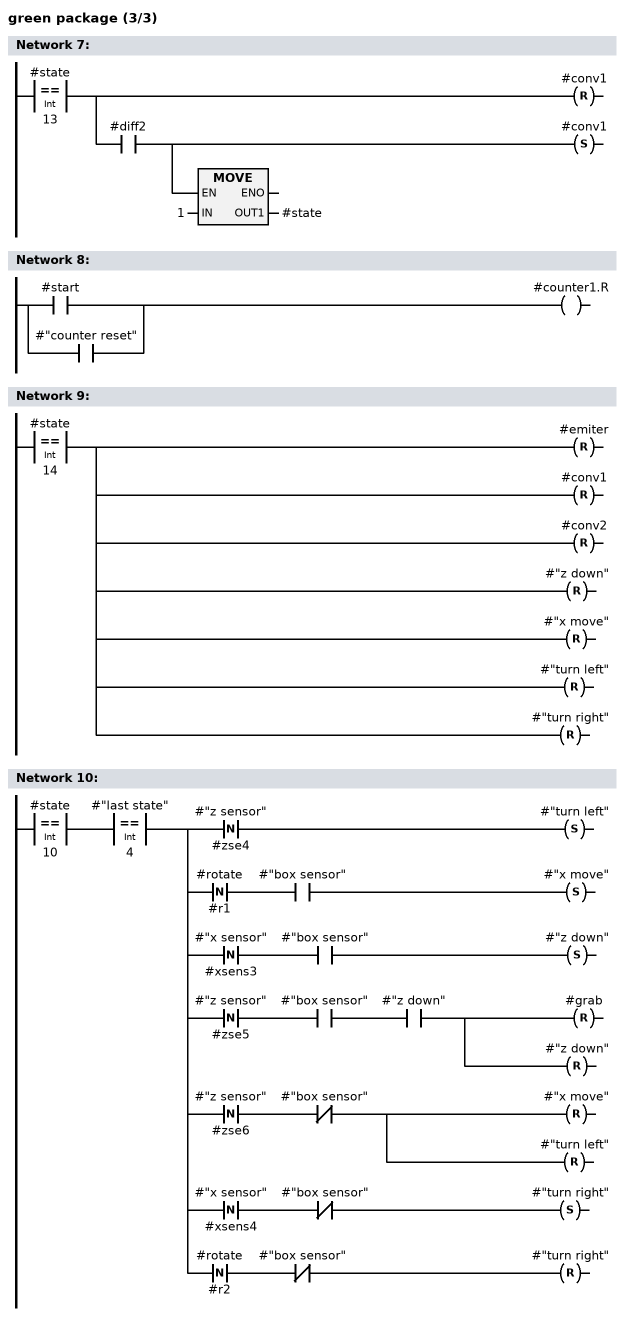
   RUNG wire#powerrail
      { S7_Templates := "SrcType := Int" } EQ_Contact(in1 := #state, in2 := 13)
      wire#w1
      R_Coil( #conv1 )
   END_RUNG
   RUNG wire#w1
      Contact( #diff2 )
      wire#w2
      S_Coil( #conv1 )
   END_RUNG
   RUNG wire#w2
      Move(in := 1, out1 => #state)
   END_RUNG
   // the same network as SCL:
   #_w1 := #state = 13;
   IF #_w1 THEN #conv1 := FALSE; END_IF;
   IF #_w1 AND #diff2 THEN
       #conv1 := TRUE;
       #state := 1;
   END_IF;
END_REGION

REGION Network 8
   RUNG wire#powerrail
      Contact( #start )
      wire#w1
      Coil( #counter1.R )
   END_RUNG
   RUNG wire#powerrail
      Contact( #"counter reset" )
   END_RUNG wire#w1
   // the same network as SCL:
   #counter1.R := #start OR #"counter reset";
END_REGION

REGION Network 9
   RUNG wire#powerrail
      { S7_Templates := "SrcType := Int" } EQ_Contact(in1 := #state, in2 := 14)
      wire#w1
      R_Coil( #emiter )
   END_RUNG
   RUNG wire#w1
      R_Coil( #conv1 )
   END_RUNG
   RUNG wire#w1
      R_Coil( #conv2 )
   END_RUNG
   RUNG wire#w1
      R_Coil( #"z down" )
   END_RUNG
   RUNG wire#w1
      R_Coil( #"x move" )
   END_RUNG
   RUNG wire#w1
      R_Coil( #"turn left" )
   END_RUNG
   RUNG wire#w1
      R_Coil( #"turn right" )
   END_RUNG
   // the same network as SCL:
   IF #state = 14 THEN
       #emiter := FALSE;
       #conv1 := FALSE;
       #conv2 := FALSE;
       #"z down" := FALSE;
       #"x move" := FALSE;
       #"turn left" := FALSE;
       #"turn right" := FALSE;
   END_IF;
END_REGION

REGION Network 10
   RUNG wire#powerrail
      { S7_Templates := "SrcType := Int" } EQ_Contact(in1 := #state, in2 := 10)
      { S7_Templates := "SrcType := Int" } EQ_Contact(in1 := #"last state", in2 := 4)
      wire#w1
      N_Contact(operand := #"z sensor", bit := #zse4)
      S_Coil( #"turn left" )
   END_RUNG
   RUNG wire#w1
      N_Contact(operand := #rotate, bit := #r1)
      Contact( #"box sensor" )
      S_Coil( #"x move" )
   END_RUNG
   RUNG wire#w1
      N_Contact(operand := #"x sensor", bit := #xsens3)
      Contact( #"box sensor" )
      S_Coil( #"z down" )
   END_RUNG
   RUNG wire#w1
      N_Contact(operand := #"z sensor", bit := #zse5)
      Contact( #"box sensor" )
      Contact( #"z down" )
      wire#w2
      R_Coil( #grab )
   END_RUNG
   RUNG wire#w2
      R_Coil( #"z down" )
   END_RUNG
   RUNG wire#w1
      N_Contact(operand := #"z sensor", bit := #zse6)
      I_Contact( #"box sensor" )
      wire#w3
      R_Coil( #"x move" )
   END_RUNG
   RUNG wire#w3
      R_Coil( #"turn left" )
   END_RUNG
   RUNG wire#w1
      N_Contact(operand := #"x sensor", bit := #xsens4)
      I_Contact( #"box sensor" )
      S_Coil( #"turn right" )
   END_RUNG
   RUNG wire#w1
      N_Contact(operand := #rotate, bit := #r2)
      I_Contact( #"box sensor" )
      R_Coil( #"turn right" )
   END_RUNG
   // the same network as SCL:
   #_w1 := (#state = 10) AND (#"last state" = 4);
   #_w2 := #_w1 AND NOT #"z sensor" AND #zse4;   // falling edge of #"z sensor"
   #zse4 := #"z sensor";
   IF #_w2 THEN #"turn left" := TRUE; END_IF;
   #_w3 := #_w1 AND NOT #rotate AND #r1;   // falling edge of #rotate
   #r1 := #rotate;
   IF #_w3 AND #"box sensor" THEN #"x move" := TRUE; END_IF;
   #_w4 := #_w1 AND NOT #"x sensor" AND #xsens3;   // falling edge of #"x sensor"
   #xsens3 := #"x sensor";
   IF #_w4 AND #"box sensor" THEN #"z down" := TRUE; END_IF;
   #_w5 := #_w1 AND NOT #"z sensor" AND #zse5;   // falling edge of #"z sensor"
   #zse5 := #"z sensor";
   IF #_w5 AND #"box sensor" AND #"z down" THEN
       #grab := FALSE;
       #"z down" := FALSE;
   END_IF;
   #_w6 := #_w1 AND NOT #"z sensor" AND #zse6;   // falling edge of #"z sensor"
   #zse6 := #"z sensor";
   IF #_w6 AND NOT #"box sensor" THEN
       #"x move" := FALSE;
       #"turn left" := FALSE;
   END_IF;
   #_w7 := #_w1 AND NOT #"x sensor" AND #xsens4;   // falling edge of #"x sensor"
   #xsens4 := #"x sensor";
   IF #_w7 AND NOT #"box sensor" THEN #"turn right" := TRUE; END_IF;
   #_w8 := #_w1 AND NOT #rotate AND #r2;   // falling edge of #rotate
   #r2 := #rotate;
   IF #_w8 AND NOT #"box sensor" THEN #"turn right" := FALSE; END_IF;
END_REGION
END_FUNCTION_BLOCK

FUNCTION_BLOCK "start conver"   // FB6, LAD
{ S7_Optimized_Access := 'TRUE' }
VERSION : 0.1
   VAR_INPUT
      start : Bool;
      stop : Bool;
      emergency : Bool;
   END_VAR
   VAR_OUTPUT
      c1 : Bool;
      c2 : Bool;
      c3 : Bool;
      c4 : Bool;
      c5 : Bool;
      c6 : Bool;
      c7 : Bool;
      c8 : Bool;
      c11 : Bool;
      c12 : Bool;
      c13 : Bool;
      "counter reset" : Bool;
   END_VAR
   VAR
      countr : "counters";
   END_VAR
BEGIN

REGION Network 2
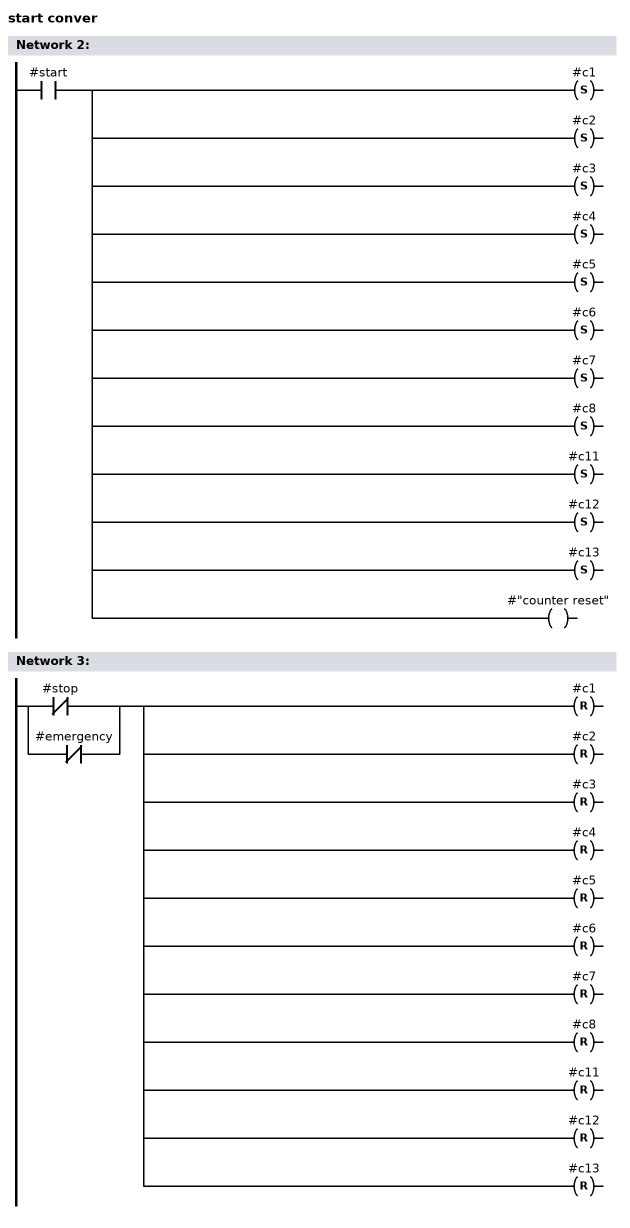
   RUNG wire#powerrail
      Contact( #start )
      wire#w1
      S_Coil( #c1 )
   END_RUNG
   RUNG wire#w1
      S_Coil( #c2 )
   END_RUNG
   RUNG wire#w1
      S_Coil( #c3 )
   END_RUNG
   RUNG wire#w1
      S_Coil( #c4 )
   END_RUNG
   RUNG wire#w1
      S_Coil( #c5 )
   END_RUNG
   RUNG wire#w1
      S_Coil( #c6 )
   END_RUNG
   RUNG wire#w1
      S_Coil( #c7 )
   END_RUNG
   RUNG wire#w1
      S_Coil( #c8 )
   END_RUNG
   RUNG wire#w1
      S_Coil( #c11 )
   END_RUNG
   RUNG wire#w1
      S_Coil( #c12 )
   END_RUNG
   RUNG wire#w1
      S_Coil( #c13 )
   END_RUNG
   RUNG wire#w1
      Coil( #"counter reset" )
   END_RUNG
   // the same network as SCL:
   IF #start THEN
       #c1 := TRUE;
       #c2 := TRUE;
       #c3 := TRUE;
       #c4 := TRUE;
       #c5 := TRUE;
       #c6 := TRUE;
       #c7 := TRUE;
       #c8 := TRUE;
       #c11 := TRUE;
       #c12 := TRUE;
       #c13 := TRUE;
   END_IF;
   #"counter reset" := #start;
END_REGION

REGION Network 3
   RUNG wire#powerrail
      I_Contact( #stop )
      wire#w1
      R_Coil( #c1 )
   END_RUNG
   RUNG wire#powerrail
      I_Contact( #emergency )
   END_RUNG wire#w1
   RUNG wire#w1
      R_Coil( #c2 )
   END_RUNG
   RUNG wire#w1
      R_Coil( #c3 )
   END_RUNG
   RUNG wire#w1
      R_Coil( #c4 )
   END_RUNG
   RUNG wire#w1
      R_Coil( #c5 )
   END_RUNG
   RUNG wire#w1
      R_Coil( #c6 )
   END_RUNG
   RUNG wire#w1
      R_Coil( #c7 )
   END_RUNG
   RUNG wire#w1
      R_Coil( #c8 )
   END_RUNG
   RUNG wire#w1
      R_Coil( #c11 )
   END_RUNG
   RUNG wire#w1
      R_Coil( #c12 )
   END_RUNG
   RUNG wire#w1
      R_Coil( #c13 )
   END_RUNG
   // the same network as SCL:
   IF NOT #stop OR NOT #emergency THEN
       #c1 := FALSE;
       #c2 := FALSE;
       #c3 := FALSE;
       #c4 := FALSE;
       #c5 := FALSE;
       #c6 := FALSE;
       #c7 := FALSE;
       #c8 := FALSE;
       #c11 := FALSE;
       #c12 := FALSE;
       #c13 := FALSE;
   END_IF;
END_REGION
END_FUNCTION_BLOCK

FUNCTION_BLOCK "palletizer"   // FB7, LAD
{ S7_Optimized_Access := 'TRUE' }
VERSION : 0.1
   VAR_INPUT
      start : Bool;
      stop : Bool;
      emergecy : Bool;
      diff : Bool;
      "pusher sensor" : Bool;
      "front limit" : Bool;
      "back limit" : Bool;
      "elevator moving" : Bool;
      "at entry" : Bool;
      "open plate senso" : Bool;
   END_VAR
   VAR_OUTPUT
      "pallet emiter" : Bool;
      "pallet conv" : Bool;
      "box emitter" : Bool;
      c1 : Bool;
      c2 : Bool;
      "load belt" : Bool;
      pusher : Bool;
      clamp : Bool;
      "move to limit" : Bool;
      "elevator+" : Bool;
      "elevator-" : Bool;
      "chain+" : Bool;
      "pallet conver out" : Bool;
      "open plate" : Bool;
   END_VAR
   VAR
      "counter" : IEC_COUNTER;
   END_VAR
   VAR RETAIN
      "pusher counter" : IEC_COUNTER;
      "pall counter" : IEC_COUNTER;
      state : Int;
   END_VAR
   VAR
      "last state" : Int;
      "diff state" : Bool;
      "timer" : IEC_TIMER;
      timer2 : IEC_TIMER;
      timer3 : IEC_TIMER;
      timer4 : IEC_TIMER;
      timer5 : IEC_TIMER;
      timer6 : IEC_TIMER;
      timer7 : IEC_TIMER;
      timer8 : IEC_TIMER;
      timer9 : IEC_TIMER;
      timer10 : IEC_TIMER;
      timer11 : IEC_TIMER;
      timer12 : IEC_TIMER;
      "counter reset" : Bool;
      "elevator moving state 1" : Bool;
      "elevator moving state 2" : Bool;
      "at entry state" : Bool;
      "front limit state" : Bool;
      arrive : Bool;
      "open plate state" : Bool;
      counter_ : IEC_COUNTER;
      "pusher counter_" : IEC_COUNTER;
      "pall counter_" : IEC_COUNTER;
      "diff state_" : Bool;
      timer_ : IEC_TIMER;
      timer2_ : IEC_TIMER;
      timer3_ : IEC_TIMER;
      timer4_ : IEC_TIMER;
      timer5_ : IEC_TIMER;
      timer6_ : IEC_TIMER;
      timer7_ : IEC_TIMER;
      "front limit state_" : Bool;
      "at entry state_" : Bool;
      "timer10 state" : Bool;
      "reset pall counter" : Bool;
      "front limit state 2" : Bool;
   END_VAR
   VAR_TEMP   // added for the SCL form of the ladder/FBD networks
      _w1 : Bool;
      _w2 : Bool;
      _w3 : Bool;
   END_VAR
   // "counter".CV := 0;
BEGIN

REGION Network 1
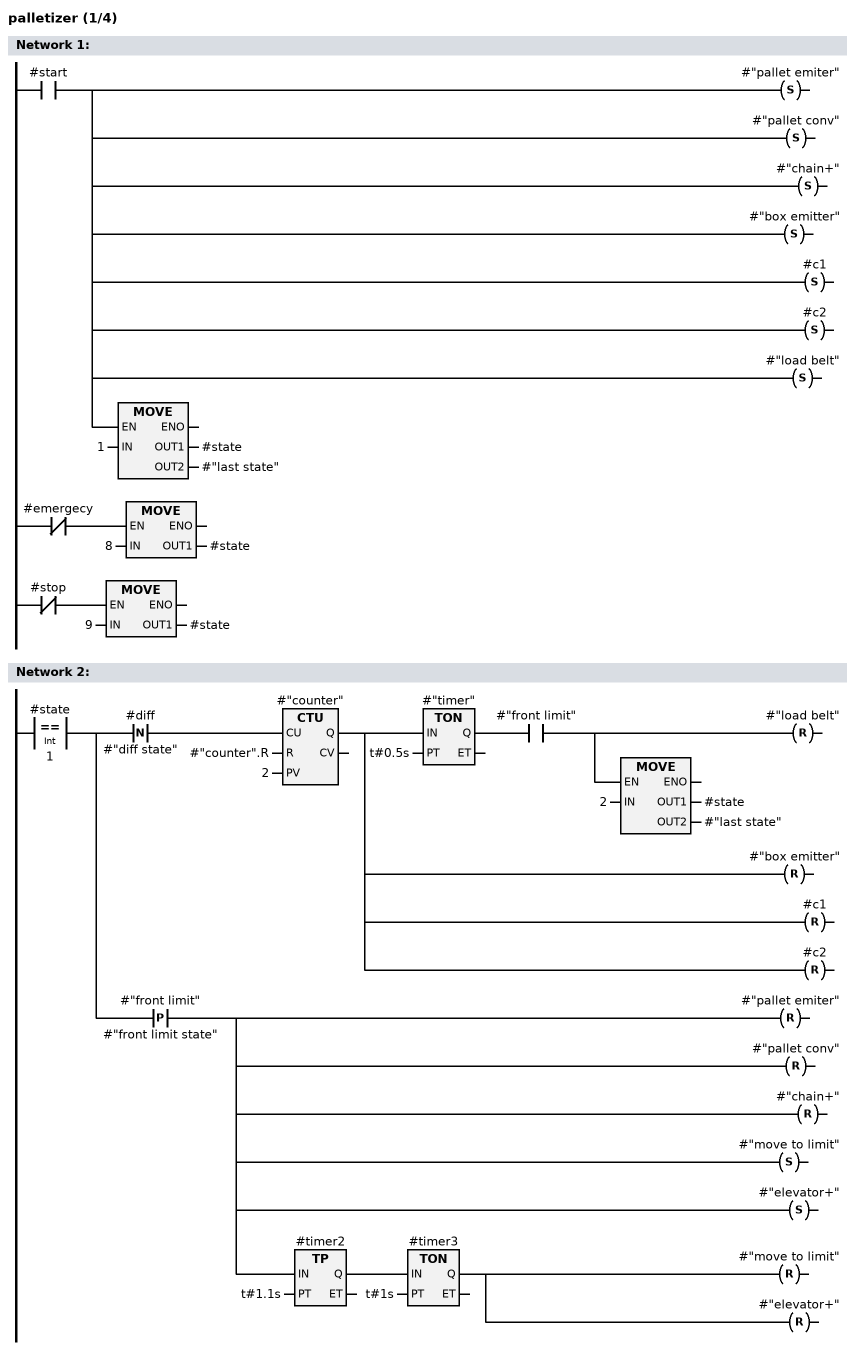
   RUNG wire#powerrail
      Contact( #start )
      wire#w1
      S_Coil( #"pallet emiter" )
   END_RUNG
   RUNG wire#w1
      S_Coil( #"pallet conv" )
   END_RUNG
   RUNG wire#w1
      S_Coil( #"chain+" )
   END_RUNG
   RUNG wire#w1
      S_Coil( #"box emitter" )
   END_RUNG
   RUNG wire#w1
      S_Coil( #c1 )
   END_RUNG
   RUNG wire#w1
      S_Coil( #c2 )
   END_RUNG
   RUNG wire#w1
      S_Coil( #"load belt" )
   END_RUNG
   RUNG wire#w1
      Move(in := 1, out1 => #state, out2 => #"last state")
   END_RUNG
   RUNG wire#powerrail
      I_Contact( #emergecy )
      Move(in := 8, out1 => #state)
   END_RUNG
   RUNG wire#powerrail
      I_Contact( #stop )
      Move(in := 9, out1 => #state)
   END_RUNG
   // the same network as SCL:
   IF #start THEN
       #"pallet emiter" := TRUE;
       #"pallet conv" := TRUE;
       #"chain+" := TRUE;
       #"box emitter" := TRUE;
       #c1 := TRUE;
       #c2 := TRUE;
       #"load belt" := TRUE;
       #state := 1;
       #"last state" := 1;
   END_IF;
   IF NOT #emergecy THEN #state := 8; END_IF;
   IF NOT #stop THEN #state := 9; END_IF;
END_REGION

REGION Network 2
   #_w1 := #state = 1;
   #_w2 := #_w1 AND NOT #diff AND #"diff state";   // falling edge of #diff
   #"diff state" := #diff;
   #"counter".CTU(CU := #_w2, R := #"counter".R, PV := 2);
   #"timer".TON(IN := #"counter".Q, PT := t#0.5s);
   IF #"timer".Q AND #"front limit" THEN
       #"load belt" := FALSE;
       #state := 2;
       #"last state" := 2;
   END_IF;
   IF #"counter".Q THEN
       #"box emitter" := FALSE;
       #c1 := FALSE;
       #c2 := FALSE;
   END_IF;
   #_w3 := #_w1 AND #"front limit" AND NOT #"front limit state";   // rising edge of #"front limit"
   #"front limit state" := #"front limit";
   IF #_w3 THEN
       #"pallet emiter" := FALSE;
       #"pallet conv" := FALSE;
       #"chain+" := FALSE;
       #"move to limit" := TRUE;
       #"elevator+" := TRUE;
   END_IF;
   #timer2.TP(IN := #_w3, PT := t#1.1s);
   #timer3.TON(IN := #timer2.Q, PT := t#1s);
   IF #timer3.Q THEN
       #"move to limit" := FALSE;
       #"elevator+" := FALSE;
   END_IF;
END_REGION

REGION Network 3
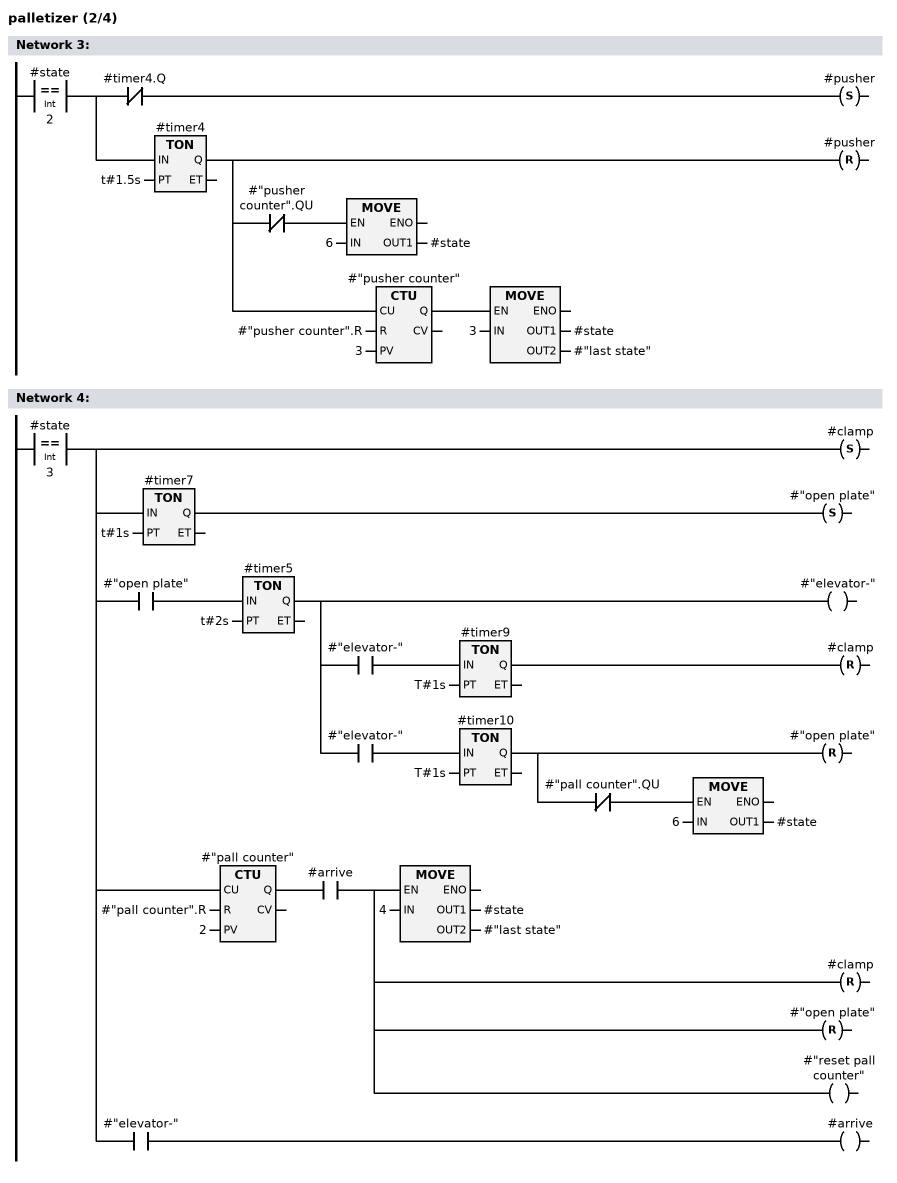
   #_w1 := #state = 2;
   IF #_w1 AND NOT #timer4.Q THEN #pusher := TRUE; END_IF;
   #timer4.TON(IN := #_w1, PT := t#1.5s);
   IF #timer4.Q THEN #pusher := FALSE; END_IF;
   IF #timer4.Q AND NOT #"pusher counter".QU THEN #state := 6; END_IF;
   #"pusher counter".CTU(CU := #timer4.Q, R := #"pusher counter".R, PV := 3);
   IF #"pusher counter".Q THEN
       #state := 3;
       #"last state" := 3;
   END_IF;
END_REGION

REGION Network 4
   #_w1 := #state = 3;
   IF #_w1 THEN #clamp := TRUE; END_IF;
   #timer7.TON(IN := #_w1, PT := t#1s);
   IF #timer7.Q THEN #"open plate" := TRUE; END_IF;
   #timer5.TON(IN := #_w1 AND #"open plate", PT := t#2s);
   #"elevator-" := #timer5.Q;
   #timer9.TON(IN := #timer5.Q AND #"elevator-", PT := T#1s);
   IF #timer9.Q THEN #clamp := FALSE; END_IF;
   #timer10.TON(IN := #timer5.Q AND #"elevator-", PT := T#1s);
   IF #timer10.Q THEN #"open plate" := FALSE; END_IF;
   IF #timer10.Q AND NOT #"pall counter".QU THEN #state := 6; END_IF;
   #"pall counter".CTU(CU := #_w1, R := #"pall counter".R, PV := 2);
   #_w2 := #"pall counter".Q AND #arrive;
   IF #_w2 THEN
       #state := 4;
       #"last state" := 4;
       #clamp := FALSE;
       #"open plate" := FALSE;
   END_IF;
   #"reset pall counter" := #_w2;
   #arrive := #_w1 AND #"elevator-";
END_REGION

REGION Network 5
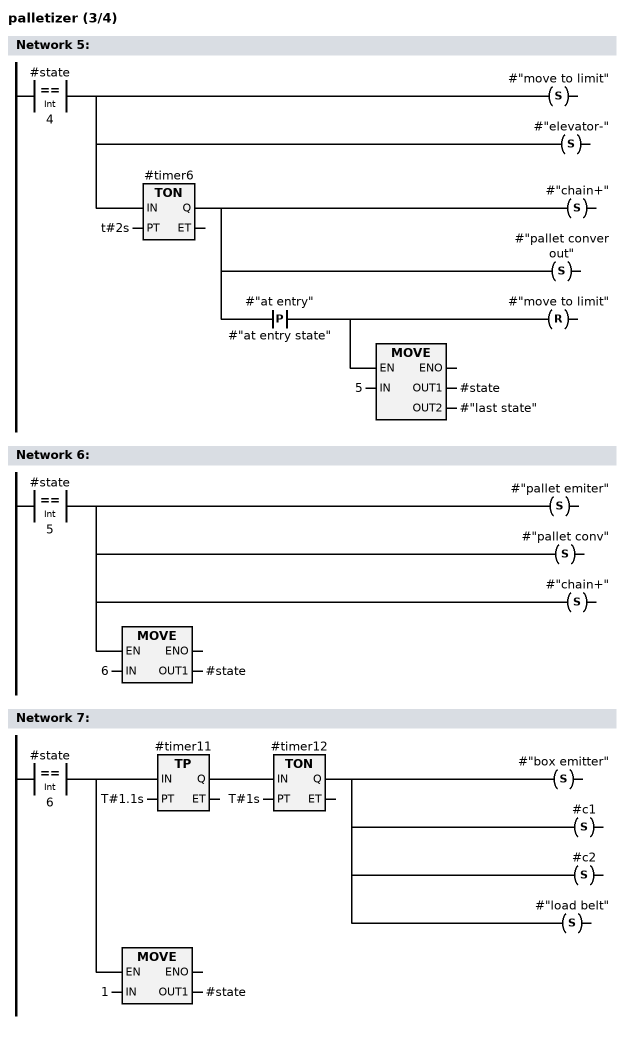
   #_w1 := #state = 4;
   IF #_w1 THEN
       #"move to limit" := TRUE;
       #"elevator-" := TRUE;
   END_IF;
   #timer6.TON(IN := #_w1, PT := t#2s);
   IF #timer6.Q THEN
       #"chain+" := TRUE;
       #"pallet conver out" := TRUE;
   END_IF;
   #_w2 := #timer6.Q AND #"at entry" AND NOT #"at entry state";   // rising edge of #"at entry"
   #"at entry state" := #"at entry";
   IF #_w2 THEN
       #"move to limit" := FALSE;
       #state := 5;
       #"last state" := 5;
   END_IF;
END_REGION

REGION Network 6
   RUNG wire#powerrail
      { S7_Templates := "SrcType := Int" } EQ_Contact(in1 := #state, in2 := 5)
      wire#w1
      S_Coil( #"pallet emiter" )
   END_RUNG
   RUNG wire#w1
      S_Coil( #"pallet conv" )
   END_RUNG
   RUNG wire#w1
      S_Coil( #"chain+" )
   END_RUNG
   RUNG wire#w1
      Move(in := 6, out1 => #state)
   END_RUNG
   // the same network as SCL:
   IF #state = 5 THEN
       #"pallet emiter" := TRUE;
       #"pallet conv" := TRUE;
       #"chain+" := TRUE;
       #state := 6;
   END_IF;
END_REGION

REGION Network 7
   #_w1 := #state = 6;
   #timer11.TP(IN := #_w1, PT := T#1.1s);
   #timer12.TON(IN := #timer11.Q, PT := T#1s);
   IF #timer12.Q THEN
       #"box emitter" := TRUE;
       #c1 := TRUE;
       #c2 := TRUE;
       #"load belt" := TRUE;
   END_IF;
   IF #_w1 THEN #state := 1; END_IF;
END_REGION

REGION Network 8
   // counter reset
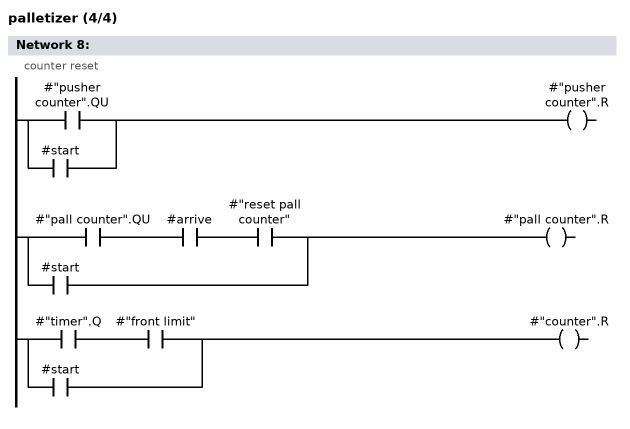
   RUNG wire#powerrail
      Contact( #"pusher counter".QU )
      wire#w1
      Coil( #"pusher counter".R )
   END_RUNG
   RUNG wire#powerrail
      Contact( #start )
   END_RUNG wire#w1
   RUNG wire#powerrail
      Contact( #"pall counter".QU )
      Contact( #arrive )
      Contact( #"reset pall counter" )
      wire#w2
      Coil( #"pall counter".R )
   END_RUNG
   RUNG wire#powerrail
      Contact( #start )
   END_RUNG wire#w2
   RUNG wire#powerrail
      Contact( #"timer".Q )
      Contact( #"front limit" )
      wire#w3
      Coil( #"counter".R )
   END_RUNG
   RUNG wire#powerrail
      Contact( #start )
   END_RUNG wire#w3
   // the same network as SCL:
   #"pusher counter".R := #"pusher counter".QU OR #start;
   #"pall counter".R := (#"pall counter".QU AND #arrive AND #"reset pall counter") OR #start;
   #"counter".R := (#"timer".Q AND #"front limit") OR #start;
END_REGION
END_FUNCTION_BLOCK

FUNCTION_BLOCK "turn table"   // FB8, LAD
{ S7_Optimized_Access := 'TRUE' }
VERSION : 0.1
   VAR_INPUT
      "line entry g" : Bool;
      "line exit g" : Bool;
      "line entry b" : Bool;
      "line exit b" : Bool;
      "front limit" : Bool;
      "limit 90" : Bool;
      "limit 0" : Bool;
      "line exit finished" : Bool;
   END_VAR
   VAR_OUTPUT
      ci1g : Bool;
      ci2g : Bool;
      ci1b : Bool;
      ci2b : Bool;
      ci3b : Bool;
      rsg : Bool;
      rsb : Bool;
      "roll+" : Bool;
      "roll-" : Bool;
      "turn table+" : Bool;
      "turn table-" : Bool;
      co1 : Bool;
   END_VAR
   VAR
      state : Int;
      "state green" : Int;
      "state blue" : Int;
      ctu1 : IEC_UCOUNTER;
      ctu2 : IEC_UCOUNTER;
   END_VAR
   VAR RETAIN
      "line entry state g" : Bool;
   END_VAR
   VAR
      "line entry state g_1" : Bool;
      "line entry state b" : Bool;
      "line entry state b_1" : Bool;
      "line exit state g" : Bool;
      "line exit finished state 1 g" : Bool;
      "line exit state b" : Bool;
      "line exit state b_1" : Bool;
      "front limit state g" : Bool;
      "front limit state b" : Bool;
      "line exit finished state g" : Bool;
      "line exit finished state b" : Bool;
      "limit 0 state g" : Bool;
      "limit 0 state 1 g" : Bool;
      "limit 0 state b" : Bool;
      "limit 90 state b" : Bool;
      "timer" : IEC_TIMER;
      timer1 : IEC_TIMER;
      timer2 : IEC_TIMER;
   END_VAR
   VAR_TEMP   // added for the SCL form of the ladder/FBD networks
      _w1 : Bool;
      _w2 : Bool;
      _w3 : Bool;
      _w4 : Bool;
      _w5 : Bool;
   END_VAR
BEGIN

REGION Network 2
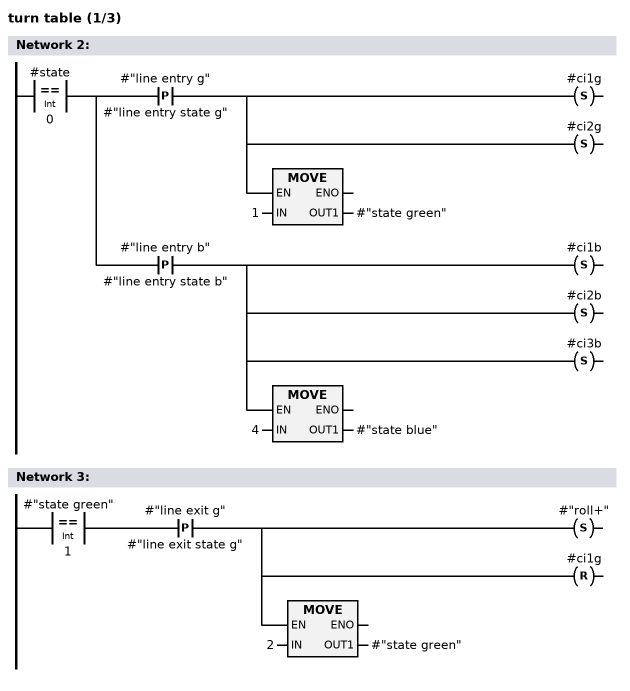
   RUNG wire#powerrail
      { S7_Templates := "SrcType := Int" } EQ_Contact(in1 := #state, in2 := 0)
      wire#w1
      P_Contact(operand := #"line entry g", bit := #"line entry state g")
      wire#w2
      S_Coil( #ci1g )
   END_RUNG
   RUNG wire#w2
      S_Coil( #ci2g )
   END_RUNG
   RUNG wire#w2
      Move(in := 1, out1 => #"state green")
   END_RUNG
   RUNG wire#w1
      P_Contact(operand := #"line entry b", bit := #"line entry state b")
      wire#w3
      S_Coil( #ci1b )
   END_RUNG
   RUNG wire#w3
      S_Coil( #ci2b )
   END_RUNG
   RUNG wire#w3
      S_Coil( #ci3b )
   END_RUNG
   RUNG wire#w3
      Move(in := 4, out1 => #"state blue")
   END_RUNG
   // the same network as SCL:
   #_w1 := #state = 0;
   #_w2 := #_w1 AND #"line entry g" AND NOT #"line entry state g";   // rising edge of #"line entry g"
   #"line entry state g" := #"line entry g";
   IF #_w2 THEN
       #ci1g := TRUE;
       #ci2g := TRUE;
       #"state green" := 1;
   END_IF;
   #_w3 := #_w1 AND #"line entry b" AND NOT #"line entry state b";   // rising edge of #"line entry b"
   #"line entry state b" := #"line entry b";
   IF #_w3 THEN
       #ci1b := TRUE;
       #ci2b := TRUE;
       #ci3b := TRUE;
       #"state blue" := 4;
   END_IF;
END_REGION

REGION Network 3
   RUNG wire#powerrail
      { S7_Templates := "SrcType := Int" } EQ_Contact(in1 := #"state green", in2 := 1)
      P_Contact(operand := #"line exit g", bit := #"line exit state g")
      wire#w1
      S_Coil( #"roll+" )
   END_RUNG
   RUNG wire#w1
      R_Coil( #ci1g )
   END_RUNG
   RUNG wire#w1
      Move(in := 2, out1 => #"state green")
   END_RUNG
   // the same network as SCL:
   #_w1 := (#"state green" = 1) AND #"line exit g" AND NOT #"line exit state g";   // rising edge of #"line exit g"
   #"line exit state g" := #"line exit g";
   IF #_w1 THEN
       #"roll+" := TRUE;
       #ci1g := FALSE;
       #"state green" := 2;
   END_IF;
END_REGION

REGION Network 4
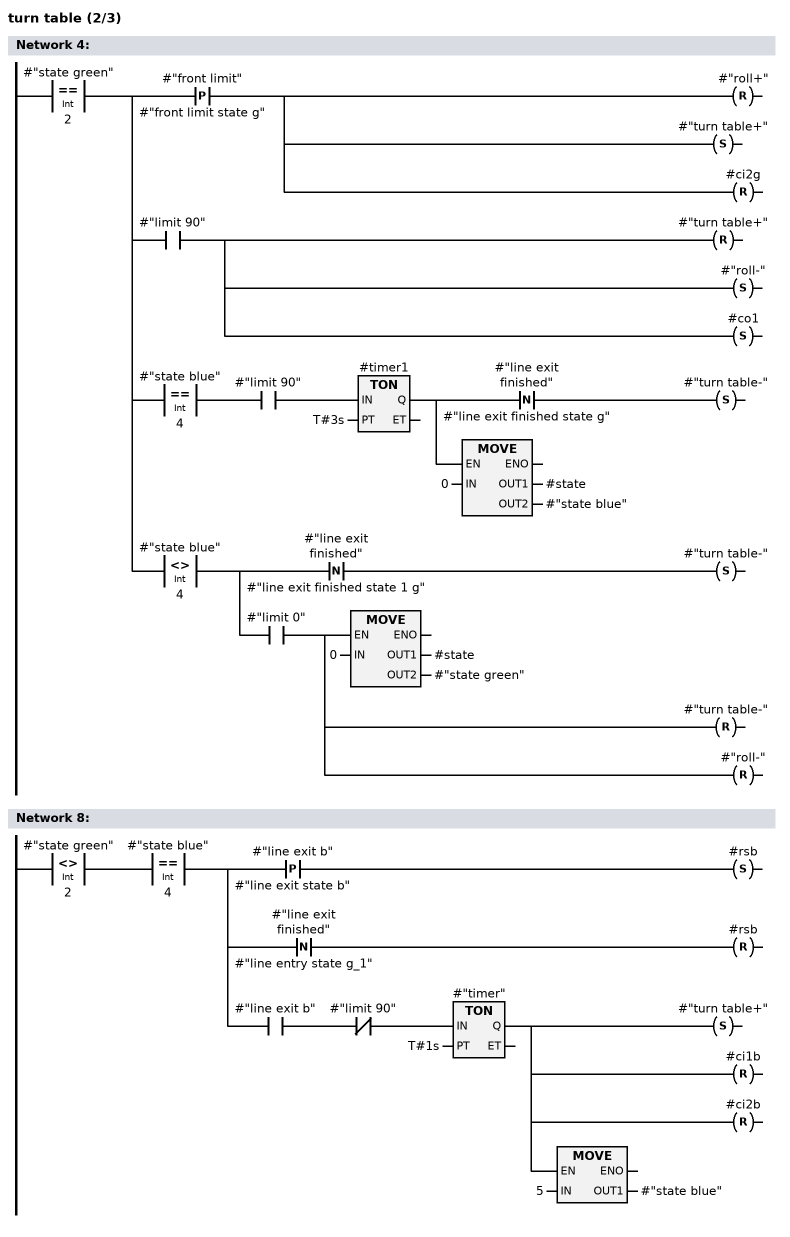
   #_w1 := #"state green" = 2;
   #_w2 := #_w1 AND #"front limit" AND NOT #"front limit state g";   // rising edge of #"front limit"
   #"front limit state g" := #"front limit";
   IF #_w2 THEN
       #"roll+" := FALSE;
       #"turn table+" := TRUE;
       #ci2g := FALSE;
   END_IF;
   IF #_w1 AND #"limit 90" THEN
       #"turn table+" := FALSE;
       #"roll-" := TRUE;
       #co1 := TRUE;
   END_IF;
   #timer1.TON(IN := #_w1 AND (#"state blue" = 4) AND #"limit 90", PT := T#3s);
   #_w3 := #timer1.Q AND NOT #"line exit finished" AND #"line exit finished state g";   // falling edge of #"line exit finished"
   #"line exit finished state g" := #"line exit finished";
   IF #_w3 THEN #"turn table-" := TRUE; END_IF;
   IF #timer1.Q THEN
       #state := 0;
       #"state blue" := 0;
   END_IF;
   #_w4 := #_w1 AND (#"state blue" <> 4);
   #_w5 := #_w4 AND NOT #"line exit finished" AND #"line exit finished state 1 g";   // falling edge of #"line exit finished"
   #"line exit finished state 1 g" := #"line exit finished";
   IF #_w5 THEN #"turn table-" := TRUE; END_IF;
   IF #_w4 AND #"limit 0" THEN
       #state := 0;
       #"state green" := 0;
       #"turn table-" := FALSE;
       #"roll-" := FALSE;
   END_IF;
END_REGION

REGION Network 8
   #_w1 := (#"state green" <> 2) AND (#"state blue" = 4);
   #_w2 := #_w1 AND #"line exit b" AND NOT #"line exit state b";   // rising edge of #"line exit b"
   #"line exit state b" := #"line exit b";
   IF #_w2 THEN #rsb := TRUE; END_IF;
   #_w3 := #_w1 AND NOT #"line exit finished" AND #"line entry state g_1";   // falling edge of #"line exit finished"
   #"line entry state g_1" := #"line exit finished";
   IF #_w3 THEN #rsb := FALSE; END_IF;
   #"timer".TON(IN := #_w1 AND #"line exit b" AND NOT #"limit 90", PT := T#1s);
   IF #"timer".Q THEN
       #"turn table+" := TRUE;
       #ci1b := FALSE;
       #ci2b := FALSE;
       #"state blue" := 5;
   END_IF;
END_REGION

REGION Network 9
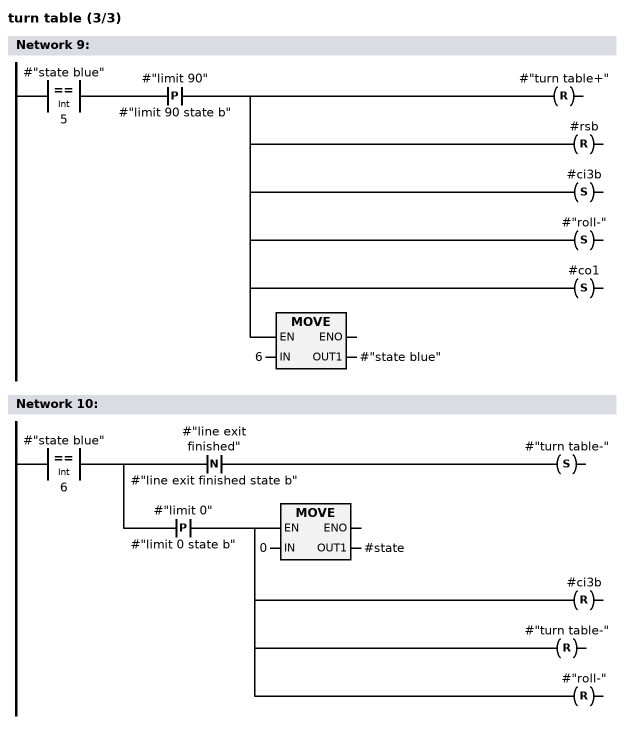
   RUNG wire#powerrail
      { S7_Templates := "SrcType := Int" } EQ_Contact(in1 := #"state blue", in2 := 5)
      P_Contact(operand := #"limit 90", bit := #"limit 90 state b")
      wire#w1
      R_Coil( #"turn table+" )
   END_RUNG
   RUNG wire#w1
      R_Coil( #rsb )
   END_RUNG
   RUNG wire#w1
      S_Coil( #ci3b )
   END_RUNG
   RUNG wire#w1
      S_Coil( #"roll-" )
   END_RUNG
   RUNG wire#w1
      S_Coil( #co1 )
   END_RUNG
   RUNG wire#w1
      Move(in := 6, out1 => #"state blue")
   END_RUNG
   // the same network as SCL:
   #_w1 := (#"state blue" = 5) AND #"limit 90" AND NOT #"limit 90 state b";   // rising edge of #"limit 90"
   #"limit 90 state b" := #"limit 90";
   IF #_w1 THEN
       #"turn table+" := FALSE;
       #rsb := FALSE;
       #ci3b := TRUE;
       #"roll-" := TRUE;
       #co1 := TRUE;
       #"state blue" := 6;
   END_IF;
END_REGION

REGION Network 10
   RUNG wire#powerrail
      { S7_Templates := "SrcType := Int" } EQ_Contact(in1 := #"state blue", in2 := 6)
      wire#w1
      N_Contact(operand := #"line exit finished", bit := #"line exit finished state b")
      S_Coil( #"turn table-" )
   END_RUNG
   RUNG wire#w1
      P_Contact(operand := #"limit 0", bit := #"limit 0 state b")
      wire#w2
      Move(in := 0, out1 => #state)
   END_RUNG
   RUNG wire#w2
      R_Coil( #ci3b )
   END_RUNG
   RUNG wire#w2
      R_Coil( #"turn table-" )
   END_RUNG
   RUNG wire#w2
      R_Coil( #"roll-" )
   END_RUNG
   // the same network as SCL:
   #_w1 := #"state blue" = 6;
   #_w2 := #_w1 AND NOT #"line exit finished" AND #"line exit finished state b";   // falling edge of #"line exit finished"
   #"line exit finished state b" := #"line exit finished";
   IF #_w2 THEN #"turn table-" := TRUE; END_IF;
   #_w3 := #_w1 AND #"limit 0" AND NOT #"limit 0 state b";   // rising edge of #"limit 0"
   #"limit 0 state b" := #"limit 0";
   IF #_w3 THEN
       #state := 0;
       #ci3b := FALSE;
       #"turn table-" := FALSE;
       #"roll-" := FALSE;
   END_IF;
END_REGION
END_FUNCTION_BLOCK

FUNCTION_BLOCK "rack"   // FB9, LAD
{ S7_Optimized_Access := 'TRUE' }
VERSION : 0.1
   VAR_INPUT
      "entry diff" : Bool;
      "stop sensor" : Bool;
      "stacker x" : Bool;
      "stacker z" : Bool;
      "stacker right limit" : Bool;
      "stacker left limit" : Bool;
      "stacker middle limit" : Bool;
   END_VAR
   VAR_OUTPUT
      cto2 : Bool;
      cto3 : Bool;
      cto4 : Bool;
      cto5 : Bool;
      cto6 : Bool;
      cto7 : Bool;
      cto8 : Bool;
      "loading conv" : Bool;
      right : Bool;
      left : Bool;
      lift : Bool;
      pos : DInt;
      alarm : Bool;
   END_VAR
   VAR
      state : Int;
      index : Int;
      id : DInt := 0;
      "warehouse data" : "warehouse";
      "entry diff state" : Bool;
      "stop sensor state" : Bool;
      "stop sensor state2" : Bool;
      "right limit state" : Bool;
      "left limit state" : Bool;
      "z state 1" : Bool;
      "middle limit state" : Bool;
      arrive : Bool;
      "arrive state" : Bool;
      "ntrig state" : Bool;
      "z state 2" : Bool;
      "middle limit state 2" : Bool;
      move : Bool;
      "move state" : Bool;
      "move 2" : Bool;
      "move 2 state" : Bool;
      "timer 1" : IEC_TIMER;
      "timer 2" : IEC_TIMER;
      "timer 3" : IEC_TIMER;
      "timer 4" : IEC_TIMER;
      "x state" : Bool;
      add : Bool;
      "add state" : Bool;
      "stop add" : Bool;
   END_VAR
   VAR_TEMP   // added for the SCL form of the ladder/FBD networks
      _w1 : Bool;
      _w2 : Bool;
      _w3 : Bool;
      _w4 : Bool;
      _w5 : Bool;
   END_VAR
BEGIN

REGION Network 1
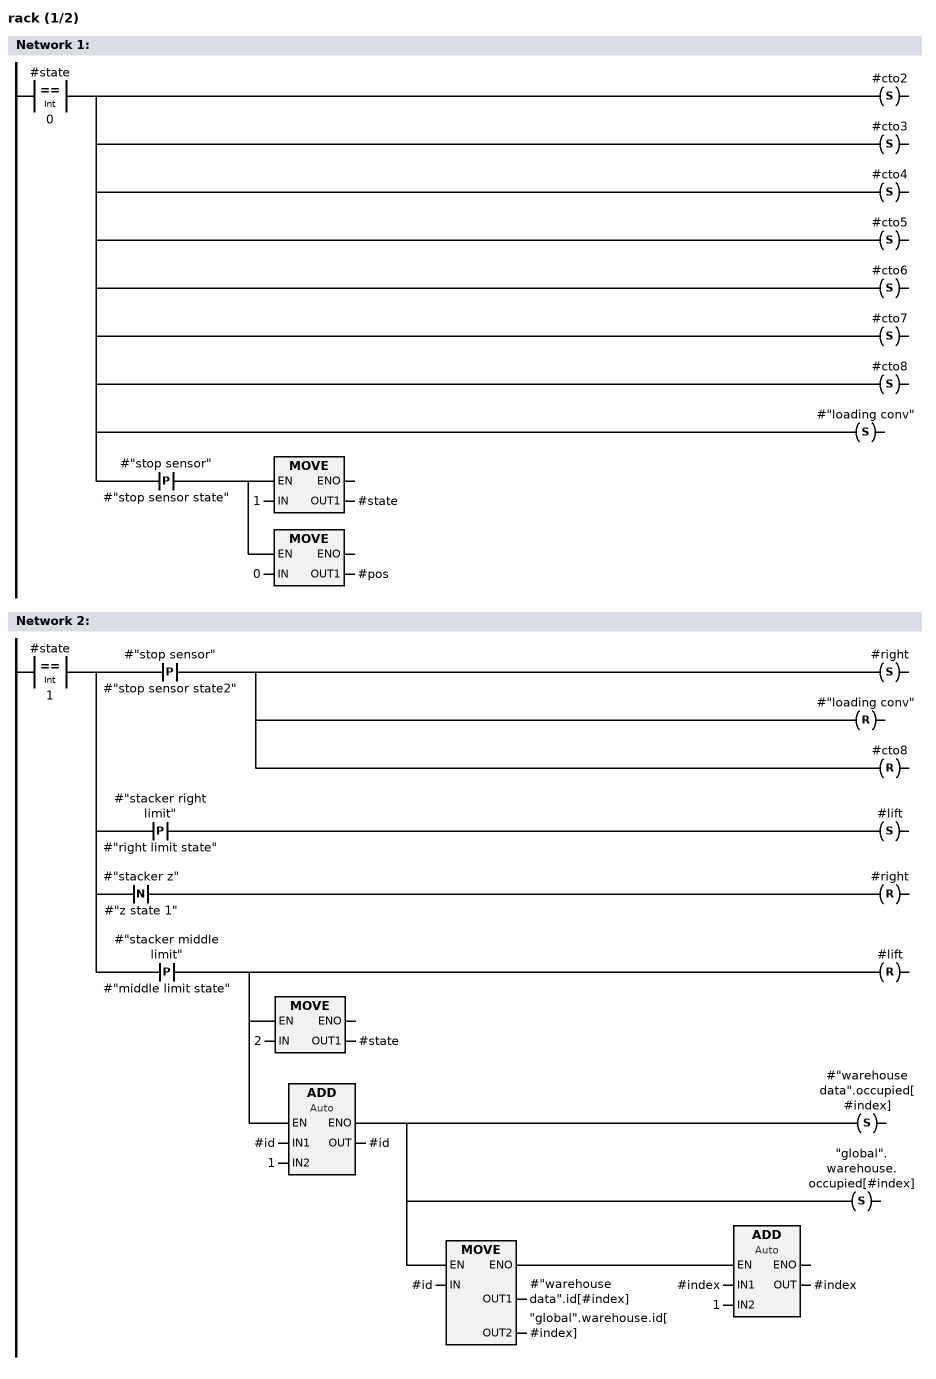
   RUNG wire#powerrail
      { S7_Templates := "SrcType := Int" } EQ_Contact(in1 := #state, in2 := 0)
      wire#w1
      S_Coil( #cto2 )
   END_RUNG
   RUNG wire#w1
      S_Coil( #cto3 )
   END_RUNG
   RUNG wire#w1
      S_Coil( #cto4 )
   END_RUNG
   RUNG wire#w1
      S_Coil( #cto5 )
   END_RUNG
   RUNG wire#w1
      S_Coil( #cto6 )
   END_RUNG
   RUNG wire#w1
      S_Coil( #cto7 )
   END_RUNG
   RUNG wire#w1
      S_Coil( #cto8 )
   END_RUNG
   RUNG wire#w1
      S_Coil( #"loading conv" )
   END_RUNG
   RUNG wire#w1
      P_Contact(operand := #"stop sensor", bit := #"stop sensor state")
      wire#w2
      Move(in := 1, out1 => #state)
   END_RUNG
   RUNG wire#w2
      Move(in := 0, out1 => #pos)
   END_RUNG
   // the same network as SCL:
   #_w1 := #state = 0;
   IF #_w1 THEN
       #cto2 := TRUE;
       #cto3 := TRUE;
       #cto4 := TRUE;
       #cto5 := TRUE;
       #cto6 := TRUE;
       #cto7 := TRUE;
       #cto8 := TRUE;
       #"loading conv" := TRUE;
   END_IF;
   #_w2 := #_w1 AND #"stop sensor" AND NOT #"stop sensor state";   // rising edge of #"stop sensor"
   #"stop sensor state" := #"stop sensor";
   IF #_w2 THEN
       #state := 1;
       #pos := 0;
   END_IF;
END_REGION

REGION Network 2
   RUNG wire#powerrail
      { S7_Templates := "SrcType := Int" } EQ_Contact(in1 := #state, in2 := 1)
      wire#w1
      P_Contact(operand := #"stop sensor", bit := #"stop sensor state2")
      wire#w2
      S_Coil( #right )
   END_RUNG
   RUNG wire#w2
      R_Coil( #"loading conv" )
   END_RUNG
   RUNG wire#w2
      R_Coil( #cto8 )
   END_RUNG
   RUNG wire#w1
      P_Contact(operand := #"stacker right limit", bit := #"right limit state")
      S_Coil( #lift )
   END_RUNG
   RUNG wire#w1
      N_Contact(operand := #"stacker z", bit := #"z state 1")
      R_Coil( #right )
   END_RUNG
   RUNG wire#w1
      P_Contact(operand := #"stacker middle limit", bit := #"middle limit state")
      wire#w3
      R_Coil( #lift )
   END_RUNG
   RUNG wire#w3
      Move(in := 2, out1 => #state)
   END_RUNG
   RUNG wire#w3
      Add(in1 := #id, in2 := 1, out => #id)
      wire#w4
      S_Coil( #"warehouse data".occupied[#index] )
   END_RUNG
   RUNG wire#w4
      S_Coil( "global".warehouse.occupied[#index] )
   END_RUNG
   RUNG wire#w4
      Move(in := #id, out1 => #"warehouse data".id[#index], out2 => "global".warehouse.id[#index])
      Add(in1 := #index, in2 := 1, out => #index)
   END_RUNG
   // the same network as SCL:
   #_w1 := #state = 1;
   #_w2 := #_w1 AND #"stop sensor" AND NOT #"stop sensor state2";   // rising edge of #"stop sensor"
   #"stop sensor state2" := #"stop sensor";
   IF #_w2 THEN
       #right := TRUE;
       #"loading conv" := FALSE;
       #cto8 := FALSE;
   END_IF;
   #_w3 := #_w1 AND #"stacker right limit" AND NOT #"right limit state";   // rising edge of #"stacker right limit"
   #"right limit state" := #"stacker right limit";
   IF #_w3 THEN #lift := TRUE; END_IF;
   #_w4 := #_w1 AND NOT #"stacker z" AND #"z state 1";   // falling edge of #"stacker z"
   #"z state 1" := #"stacker z";
   IF #_w4 THEN #right := FALSE; END_IF;
   #_w5 := #_w1 AND #"stacker middle limit" AND NOT #"middle limit state";   // rising edge of #"stacker middle limit"
   #"middle limit state" := #"stacker middle limit";
   IF #_w5 THEN
       #lift := FALSE;
       #state := 2;
       #id := #id + 1;
       #"warehouse data".occupied[#index] := TRUE;
       "global".warehouse.occupied[#index] := TRUE;
       #"warehouse data".id[#index] := #id;
       "global".warehouse.id[#index] := #id;
       #index := #index + 1;
   END_IF;
END_REGION

REGION Network 3
